LIN {X 0,Y 573.201,Z 603.99,A -85,B 0,C 180,E1 -2258.283,E2 -2258.283} C_VEL
LIN {X 0,Y 573.286,Z 595.539,A -85,B 0,C 180,E1 -2259.17,E2 -2259.17} C_VEL
LIN {X 0,Y 573.421,Z 585.099,A -85,B 0,C 180,E1 -2260.058,E2 -2260.058} C_VEL
LIN {X 0,Y 573.55,Z 573.353,A -85,B 0,C 180,E1 -2260.858,E2 -2260.858} C_VEL
LIN {X 0,Y 573.653,Z 562.283,A -85,B 0,C 180,E1 -2261.447,E2 -2261.447} C_VEL
LIN {X 0,Y 573.759,Z 549.174,A -85,B 0,C 180,E1 -2261.974,E2 -2261.974} C_VEL
LIN {X 0,Y 573.841,Z 536.522,A -85,B 0,C 180,E1 -2262.331,E2 -2262.331} C_VEL
LIN {X 0,Y 573.932,Z 523.316,A -85,B 0,C 180,E1 -2262.554,E2 -2262.554} C_VEL
LIN {X 0,Y 574.025,Z 427.51,A -85,B 0,C 180,E1 -2263.757,E2 -2263.757} C_VEL
LIN {X 0,Y 573.376,Z 423.284,A -85,B 0,C 180,E1 -2263.851,E2 -2263.851} C_VEL
LIN {X 0,Y 573.504,Z 405.17,A -85,B 0,C 180,E1 -2266.547,E2 -2266.547} C_VEL
LIN {X 0,Y 573.685,Z 388.232,A -85,B 0,C 180,E1 -2269.129,E2 -2269.129} C_VEL
LIN {X 0,Y 573.876,Z 371.34,A -85,B 0,C 180,E1 -2271.744,E2 -2271.744} C_VEL
LIN {X 0,Y 573.288,Z 367.673,A -85,B 0,C 180,E1 -2272.383,E2 -2272.383} C_VEL
LIN {X 0,Y 573.259,Z 367.581,A -85,B 0,C 180,E1 -2275.409,E2 -2275.409} C_VEL
LIN {X 0,Y 573.252,Z 367.576,A -85,B 0,C 180,E1 -2278.028,E2 -2278.028} C_VEL
LIN {X 0,Y 573.24,Z 367.576,A -85,B 0,C 180,E1 -2280.884,E2 -2280.884} C_VEL
LIN {X 0,Y 573.262,Z 367.58,A -85,B 0,C 180,E1 -2283.523,E2 -2283.523} C_VEL
LIN {X 0,Y 573.262,Z 367.573,A -85,B 0,C 180,E1 -2286.047,E2 -2286.047} C_VEL
LIN {X 0,Y 573.249,Z 367.575,A -85,B 0,C 180,E1 -2288.7,E2 -2288.7} C_VEL
LIN {X 0,Y 573.253,Z 367.577,A -85,B 0,C 180,E1 -2291.595,E2 -2291.595} C_VEL
LIN {X 0,Y 573.237,Z 367.575,A -85,B 0,C 180,E1 -2294.332,E2 -2294.332} C_VEL
LIN {X 0,Y 573.249,Z 367.58,A -85,B 0,C 180,E1 -2297.357,E2 -2297.357} C_VEL
LIN {X 0,Y 573.271,Z 367.575,A -85,B 0,C 180,E1 -2299.477,E2 -2299.477} C_VEL
LIN {X 0,Y 573.234,Z 367.575,A -85,B 0,C 180,E1 -2302.192,E2 -2302.192} C_VEL
LIN {X 0,Y 573.264,Z 367.578,A -85,B 0,C 180,E1 -2304.816,E2 -2304.816} C_VEL
LIN {X 0,Y 573.253,Z 367.577,A -85,B 0,C 180,E1 -2307.355,E2 -2307.355} C_VEL
LIN {X 0,Y 573.245,Z 367.574,A -85,B 0,C 180,E1 -2309.824,E2 -2309.824} C_VEL
LIN {X 0,Y 573.284,Z 367.571,A -85,B 0,C 180,E1 -2312.235,E2 -2312.235} C_VEL
LIN {X 0,Y 573.263,Z 367.577,A -85,B 0,C 180,E1 -2315.121,E2 -2315.121} C_VEL
LIN {X 0,Y 573.233,Z 367.576,A -85,B 0,C 180,E1 -2317.662,E2 -2317.662} C_VEL
LIN {X 0,Y 573.251,Z 367.574,A -85,B 0,C 180,E1 -2319.923,E2 -2319.923} C_VEL
LIN {X 0,Y 573.258,Z 367.578,A -85,B 0,C 180,E1 -2322.988,E2 -2322.988} C_VEL
LIN {X 0,Y 573.266,Z 367.572,A -85,B 0,C 180,E1 -2325.807,E2 -2325.807} C_VEL
LIN {X 0,Y 573.255,Z 367.58,A -85,B 0,C 180,E1 -2328.745,E2 -2328.745} C_VEL
LIN {X 0,Y 573.284,Z 367.569,A -85,B 0,C 180,E1 -2331.54,E2 -2331.54} C_VEL
LIN {X 0,Y 573.285,Z 367.578,A -85,B 0,C 180,E1 -2334.372,E2 -2334.372} C_VEL
LIN {X 0,Y 573.302,Z 367.57,A -85,B 0,C 180,E1 -2337.892,E2 -2337.892} C_VEL
LIN {X 0,Y 573.329,Z 367.568,A -85,B 0,C 180,E1 -2340.702,E2 -2340.702} C_VEL
LIN {X 0,Y 573.235,Z 367.576,A -85,B 0,C 180,E1 -2343.514,E2 -2343.514} C_VEL
LIN {X 0,Y 573.287,Z 367.57,A -85,B 0,C 180,E1 -2345.628,E2 -2345.628} C_VEL
LIN {X 0,Y 573.284,Z 367.576,A -85,B 0,C 180,E1 -2348.459,E2 -2348.459} C_VEL
LIN {X 0,Y 573.264,Z 367.572,A -85,B 0,C 180,E1 -2351.312,E2 -2351.312} C_VEL
LIN {X 0,Y 573.267,Z 367.58,A -85,B 0,C 180,E1 -2354.193,E2 -2354.193} C_VEL
LIN {X 0,Y 573.255,Z 367.573,A -85,B 0,C 180,E1 -2357.112,E2 -2357.112} C_VEL
LIN {X 0,Y 573.252,Z 367.582,A -85,B 0,C 180,E1 -2360.077,E2 -2360.077} C_VEL
LIN {X 0,Y 573.235,Z 367.58,A -85,B 0,C 180,E1 -2362.338,E2 -2362.338} C_VEL
LIN {X 0,Y 573.247,Z 367.576,A -85,B 0,C 180,E1 -2364.398,E2 -2364.398} C_VEL
LIN {X 0,Y 572.62,Z 367.654,A -85,B 0,C 180,E1 -2364.985,E2 -2364.985} C_VEL
LIN {X 0,Y 569.781,Z 368.014,A -85,B 0,C 180,E1 -2365.936,E2 -2365.936} C_VEL
LIN {X 0,Y 567.353,Z 368.314,A -85,B 0,C 180,E1 -2366.702,E2 -2366.702} C_VEL
LIN {X 0,Y 566.301,Z 368.442,A -85,B 0,C 180,E1 -2367.294,E2 -2367.294} C_VEL
LIN {X 0,Y 566.212,Z 368.452,A -85,B 0,C 180,E1 -2367.494,E2 -2367.494} C_VEL
LIN {X 0,Y 566.223,Z 368.458,A -85,B 0,C 180,E1 -2369.768,E2 -2369.768} C_VEL
LIN {X 0,Y 566.205,Z 368.453,A -85,B 0,C 180,E1 -2372.432,E2 -2372.432} C_VEL
LIN {X 0,Y 566.209,Z 368.452,A -85,B 0,C 180,E1 -2374.995,E2 -2374.995} C_VEL
LIN {X 0,Y 566.193,Z 368.459,A -85,B 0,C 180,E1 -2377.461,E2 -2377.461} C_VEL
LIN {X 0,Y 566.224,Z 368.451,A -85,B 0,C 180,E1 -2380.198,E2 -2380.198} C_VEL
LIN {X 0,Y 566.203,Z 368.454,A -85,B 0,C 180,E1 -2383.054,E2 -2383.054} C_VEL
LIN {X 0,Y 566.195,Z 368.455,A -85,B 0,C 180,E1 -2386.049,E2 -2386.049} C_VEL
LIN {X 0,Y 566.21,Z 368.452,A -85,B 0,C 180,E1 -2388.864,E2 -2388.864} C_VEL
LIN {X 0,Y 566.189,Z 368.46,A -85,B 0,C 180,E1 -2391.638,E2 -2391.638} C_VEL
LIN {X 0,Y 566.212,Z 368.45,A -85,B 0,C 180,E1 -2394.312,E2 -2394.312} C_VEL
LIN {X 0,Y 566.228,Z 368.451,A -85,B 0,C 180,E1 -2396.899,E2 -2396.899} C_VEL
LIN {X 0,Y 566.185,Z 368.461,A -85,B 0,C 180,E1 -2399.408,E2 -2399.408} C_VEL
LIN {X 0,Y 566.212,Z 368.452,A -85,B 0,C 180,E1 -2401.858,E2 -2401.858} C_VEL
LIN {X 0,Y 566.215,Z 368.45,A -85,B 0,C 180,E1 -2404.251,E2 -2404.251} C_VEL
LIN {X 0,Y 566.174,Z 368.458,A -85,B 0,C 180,E1 -2406.718,E2 -2406.718} C_VEL
LIN {X 0,Y 566.208,Z 368.452,A -85,B 0,C 180,E1 -2409.663,E2 -2409.663} C_VEL
LIN {X 0,Y 566.201,Z 368.455,A -85,B 0,C 180,E1 -2412.669,E2 -2412.669} C_VEL
LIN {X 0,Y 566.237,Z 368.449,A -85,B 0,C 180,E1 -2415.627,E2 -2415.627} C_VEL
LIN {X 0,Y 566.237,Z 368.453,A -85,B 0,C 180,E1 -2418.675,E2 -2418.675} C_VEL
LIN {X 0,Y 566.23,Z 368.454,A -85,B 0,C 180,E1 -2421.434,E2 -2421.434} C_VEL
LIN {X 0,Y 566.259,Z 368.58,A -85,B 0,C 180,E1 -2422.203,E2 -2422.203} C_VEL
LIN {X 0,Y 566.656,Z 372.244,A -85,B 0,C 180,E1 -2422.875,E2 -2422.875} C_VEL
LIN {X 0,Y 566.541,Z 387.974,A -85,B 0,C 180,E1 -2425.553,E2 -2425.553} C_VEL
LIN {X 0,Y 566.343,Z 407.089,A -85,B 0,C 180,E1 -2428.755,E2 -2428.755} C_VEL
LIN {X 0,Y 566.33,Z 408.914,A -85,B 0,C 180,E1 -2429.022,E2 -2429.022} C_VEL
LIN {X 0,Y 566.891,Z 412.581,A -85,B 0,C 180,E1 -2429.112,E2 -2429.112} C_VEL
LIN {X 0,Y 567.185,Z 418.987,A -85,B 0,C 180,E1 -2429.201,E2 -2429.201} C_VEL
LIN {X 0,Y 566.972,Z 515.705,A -85,B 0,C 180,E1 -2430.444,E2 -2430.444} C_VEL
LIN {X 0,Y 566.89,Z 528.87,A -85,B 0,C 180,E1 -2430.755,E2 -2430.755} C_VEL
LIN {X 0,Y 566.741,Z 541.512,A -85,B 0,C 180,E1 -2431.199,E2 -2431.199} C_VEL
LIN {X 0,Y 566.56,Z 553.601,A -85,B 0,C 180,E1 -2431.777,E2 -2431.777} C_VEL
LIN {X 0,Y 566.433,Z 565.04,A -85,B 0,C 180,E1 -2432.489,E2 -2432.489} C_VEL
LIN {X 0,Y 566.294,Z 575.37,A -85,B 0,C 180,E1 -2433.29,E2 -2433.29} C_VEL
LIN {X 0,Y 566.172,Z 583.857,A -85,B 0,C 180,E1 -2434.093,E2 -2434.093} C_VEL
LIN {X 0,Y 566.132,Z 591.698,A -85,B 0,C 180,E1 -2434.985,E2 -2434.985} C_VEL
LIN {X 0,Y 566.025,Z 599.41,A -85,B 0,C 180,E1 -2436.058,E2 -2436.058} C_VEL
LIN {X 0,Y 565.97,Z 605.612,A -85,B 0,C 180,E1 -2437.133,E2 -2437.133} C_VEL
LIN {X 0,Y 565.959,Z 610.553,A -85,B 0,C 180,E1 -2438.21,E2 -2438.21} C_VEL
LIN {X 0,Y 565.876,Z 614.383,A -85,B 0,C 180,E1 -2439.291,E2 -2439.291} C_VEL
LIN {X 0,Y 565.887,Z 616.355,A -85,B 0,C 180,E1 -2440.013,E2 -2440.013} C_VEL
LIN {X 0,Y 565.901,Z 618.581,A -85,B 0,C 180,E1 -2441.153,E2 -2441.153} C_VEL
LIN {X 0,Y 565.865,Z 619.69,A -85,B 0,C 180,E1 -2442.189,E2 -2442.189} C_VEL
LIN {X 0,Y 565.843,Z 619.978,A -85,B 0,C 180,E1 -2442.918,E2 -2442.918} C_VEL
LIN {X 0,Y 565.863,Z 619.855,A -85,B 0,C 180,E1 -2443.649,E2 -2443.649} C_VEL
LIN {X 0,Y 565.877,Z 619.281,A -85,B 0,C 180,E1 -2444.382,E2 -2444.382} C_VEL
LIN {X 0,Y 565.811,Z 618.293,A -85,B 0,C 180,E1 -2445.12,E2 -2445.12} C_VEL
LIN {X 0,Y 565.832,Z 616.886,A -85,B 0,C 180,E1 -2445.857,E2 -2445.857} C_VEL
LIN {X 0,Y 565.898,Z 613.759,A -85,B 0,C 180,E1 -2447.005,E2 -2447.005} C_VEL
LIN {X 0,Y 565.928,Z 609.725,A -85,B 0,C 180,E1 -2448.087,E2 -2448.087} C_VEL
LIN {X 0,Y 565.987,Z 603.691,A -85,B 0,C 180,E1 -2449.315,E2 -2449.315} C_VEL
LIN {X 0,Y 566.045,Z 596.024,A -85,B 0,C 180,E1 -2450.533,E2 -2450.533} C_VEL
LIN {X 0,Y 566.161,Z 587.806,A -85,B 0,C 180,E1 -2451.568,E2 -2451.568} C_VEL
LIN {X 0,Y 566.268,Z 578.376,A -85,B 0,C 180,E1 -2452.531,E2 -2452.531} C_VEL
LIN {X 0,Y 566.386,Z 567.954,A -85,B 0,C 180,E1 -2453.395,E2 -2453.395} C_VEL
LIN {X 0,Y 566.546,Z 556.203,A -85,B 0,C 180,E1 -2454.164,E2 -2454.164} C_VEL
LIN {X 0,Y 566.673,Z 543.843,A -85,B 0,C 180,E1 -2454.793,E2 -2454.793} C_VEL
LIN {X 0,Y 566.851,Z 531.171,A -85,B 0,C 180,E1 -2455.268,E2 -2455.268} C_VEL
LIN {X 0,Y 566.956,Z 517.562,A -85,B 0,C 180,E1 -2455.61,E2 -2455.61} C_VEL
LIN {X 0,Y 567.038,Z 490.594,A -85,B 0,C 180,E1 -2455.979,E2 -2455.979} C_VEL
LIN {X 0,Y 567.083,Z 413.826,A -85,B 0,C 180,E1 -2456.957,E2 -2456.957} C_VEL
LIN {X 0,Y 566.313,Z 409.219,A -85,B 0,C 180,E1 -2457.05,E2 -2457.05} C_VEL
LIN {X 0,Y 566.268,Z 407.096,A -85,B 0,C 180,E1 -2457.335,E2 -2457.335} C_VEL
LIN {X 0,Y 566.476,Z 390.202,A -85,B 0,C 180,E1 -2460.162,E2 -2460.162} C_VEL
LIN {X 0,Y 566.678,Z 373.075,A -85,B 0,C 180,E1 -2463.071,E2 -2463.071} C_VEL
LIN {X 0,Y 566.23,Z 368.551,A -85,B 0,C 180,E1 -2463.903,E2 -2463.903} C_VEL
LIN {X 0,Y 566.214,Z 368.453,A -85,B 0,C 180,E1 -2466.568,E2 -2466.568} C_VEL
LIN {X 0,Y 566.21,Z 368.453,A -85,B 0,C 180,E1 -2469.685,E2 -2469.685} C_VEL
LIN {X 0,Y 566.21,Z 368.451,A -85,B 0,C 180,E1 -2472.086,E2 -2472.086} C_VEL
LIN {X 0,Y 566.169,Z 368.464,A -85,B 0,C 180,E1 -2475.035,E2 -2475.035} C_VEL
LIN {X 0,Y 566.225,Z 368.447,A -85,B 0,C 180,E1 -2478.134,E2 -2478.134} C_VEL
LIN {X 0,Y 566.218,Z 368.453,A -85,B 0,C 180,E1 -2480.727,E2 -2480.727} C_VEL
LIN {X 0,Y 566.212,Z 368.45,A -85,B 0,C 180,E1 -2483.783,E2 -2483.783} C_VEL
LIN {X 0,Y 566.222,Z 368.448,A -85,B 0,C 180,E1 -2486.262,E2 -2486.262} C_VEL
LIN {X 0,Y 566.197,Z 368.46,A -85,B 0,C 180,E1 -2488.92,E2 -2488.92} C_VEL
LIN {X 0,Y 566.192,Z 368.46,A -85,B 0,C 180,E1 -2491.047,E2 -2491.047} C_VEL
LIN {X 0,Y 566.24,Z 368.449,A -85,B 0,C 180,E1 -2493.46,E2 -2493.46} C_VEL
LIN {X 0,Y 566.197,Z 368.452,A -85,B 0,C 180,E1 -2495.819,E2 -2495.819} C_VEL
LIN {X 0,Y 566.209,Z 368.458,A -85,B 0,C 180,E1 -2498.902,E2 -2498.902} C_VEL
LIN {X 0,Y 566.206,Z 368.456,A -85,B 0,C 180,E1 -2501.172,E2 -2501.172} C_VEL
LIN {X 0,Y 566.215,Z 368.452,A -85,B 0,C 180,E1 -2503.412,E2 -2503.412} C_VEL
LIN {X 0,Y 566.195,Z 368.453,A -85,B 0,C 180,E1 -2506.359,E2 -2506.359} C_VEL
LIN {X 0,Y 566.265,Z 368.449,A -85,B 0,C 180,E1 -2508.654,E2 -2508.654} C_VEL
LIN {X 0,Y 566.242,Z 368.448,A -85,B 0,C 180,E1 -2511.435,E2 -2511.435} C_VEL
LIN {X 0,Y 566.256,Z 368.445,A -85,B 0,C 180,E1 -2514.302,E2 -2514.302} C_VEL
LIN {X 0,Y 566.272,Z 368.442,A -85,B 0,C 180,E1 -2517.866,E2 -2517.866} C_VEL
LIN {X 0,Y 566.303,Z 368.446,A -85,B 0,C 180,E1 -2520.711,E2 -2520.711} C_VEL
LIN {X 0,Y 566.274,Z 368.45,A -85,B 0,C 180,E1 -2522.846,E2 -2522.846} C_VEL
LIN {X 0,Y 566.254,Z 368.444,A -85,B 0,C 180,E1 -2525.698,E2 -2525.698} C_VEL
LIN {X 0,Y 566.241,Z 368.452,A -85,B 0,C 180,E1 -2528.566,E2 -2528.566} C_VEL
LIN {X 0,Y 566.242,Z 368.447,A -85,B 0,C 180,E1 -2531.454,E2 -2531.454} C_VEL
LIN {X 0,Y 566.224,Z 368.453,A -85,B 0,C 180,E1 -2534.507,E2 -2534.507} C_VEL
LIN {X 0,Y 566.197,Z 368.452,A -85,B 0,C 180,E1 -2537.332,E2 -2537.332} C_VEL
LIN {X 0,Y 566.213,Z 368.453,A -85,B 0,C 180,E1 -2540.337,E2 -2540.337} C_VEL
LIN {X 0,Y 566.222,Z 368.449,A -85,B 0,C 180,E1 -2543.403,E2 -2543.403} C_VEL
LIN {X 0,Y 566.218,Z 368.449,A -85,B 0,C 180,E1 -2545.749,E2 -2545.749} C_VEL
LIN {X 0,Y 566.201,Z 368.454,A -85,B 0,C 180,E1 -2548.204,E2 -2548.204} C_VEL
LIN {X 0,Y 566.193,Z 368.455,A -85,B 0,C 180,E1 -2551.079,E2 -2551.079} C_VEL
LIN {X 0,Y 566.223,Z 368.448,A -85,B 0,C 180,E1 -2553.738,E2 -2553.738} C_VEL
LIN {X 0,Y 566.211,Z 368.46,A -85,B 0,C 180,E1 -2556.569,E2 -2556.569} C_VEL
LIN {X 0,Y 566.209,Z 368.45,A -85,B 0,C 180,E1 -2559.687,E2 -2559.687} C_VEL
LIN {X 0,Y 566.216,Z 368.449,A -85,B 0,C 180,E1 -2562.087,E2 -2562.087} C_VEL
LIN {X 0,Y 566.169,Z 368.457,A -85,B 0,C 180,E1 -2565.037,E2 -2565.037} C_VEL
LIN {X 0,Y 566.215,Z 368.453,A -85,B 0,C 180,E1 -2568.137,E2 -2568.137} C_VEL
LIN {X 0,Y 566.22,Z 368.455,A -85,B 0,C 180,E1 -2570.728,E2 -2570.728} C_VEL
LIN {X 0,Y 566.217,Z 368.449,A -85,B 0,C 180,E1 -2573.784,E2 -2573.784} C_VEL
LIN {X 0,Y 566.229,Z 368.454,A -85,B 0,C 180,E1 -2576.264,E2 -2576.264} C_VEL
LIN {X 0,Y 566.199,Z 368.455,A -85,B 0,C 180,E1 -2578.923,E2 -2578.923} C_VEL
LIN {X 0,Y 566.229,Z 368.45,A -85,B 0,C 180,E1 -2581.859,E2 -2581.859} C_VEL
LIN {X 0,Y 566.226,Z 368.457,A -85,B 0,C 180,E1 -2584.252,E2 -2584.252} C_VEL
LIN {X 0,Y 566.243,Z 368.528,A -85,B 0,C 180,E1 -2587.468,E2 -2587.468} C_VEL
LIN {X 0,Y 566.914,Z 372.503,A -85,B 0,C 180,E1 -2588.167,E2 -2588.167} C_VEL
LIN {X 0,Y 566.728,Z 389.583,A -85,B 0,C 180,E1 -2590.837,E2 -2590.837} C_VEL
LIN {X 0,Y 566.496,Z 406.333,A -85,B 0,C 180,E1 -2593.421,E2 -2593.421} C_VEL
LIN {X 0,Y 566.375,Z 423.296,A -85,B 0,C 180,E1 -2595.975,E2 -2595.975} C_VEL
LIN {X 0,Y 567.201,Z 430.334,A -85,B 0,C 180,E1 -2596.11,E2 -2596.11} C_VEL
LIN {X 0,Y 566.982,Z 530.968,A -85,B 0,C 180,E1 -2597.404,E2 -2597.404} C_VEL
LIN {X 0,Y 566.887,Z 544.233,A -85,B 0,C 180,E1 -2597.72,E2 -2597.72} C_VEL
LIN {X 0,Y 566.745,Z 556.386,A -85,B 0,C 180,E1 -2598.149,E2 -2598.149} C_VEL
LIN {X 0,Y 566.627,Z 568.16,A -85,B 0,C 180,E1 -2598.709,E2 -2598.709} C_VEL
LIN {X 0,Y 566.485,Z 578.914,A -85,B 0,C 180,E1 -2599.366,E2 -2599.366} C_VEL
LIN {X 0,Y 566.332,Z 589.545,A -85,B 0,C 180,E1 -2600.176,E2 -2600.176} C_VEL
LIN {X 0,Y 566.207,Z 599.116,A -85,B 0,C 180,E1 -2601.075,E2 -2601.075} C_VEL
LIN {X 0,Y 566.112,Z 606.963,A -85,B 0,C 180,E1 -2601.972,E2 -2601.972} C_VEL
LIN {X 0,Y 566.003,Z 614.624,A -85,B 0,C 180,E1 -2603.047,E2 -2603.047} C_VEL
LIN {X 0,Y 566.004,Z 621.681,A -85,B 0,C 180,E1 -2604.299,E2 -2604.299} C_VEL
LIN {X 0,Y 565.933,Z 626.373,A -85,B 0,C 180,E1 -2605.37,E2 -2605.37} C_VEL
LIN {X 0,Y 565.927,Z 629.958,A -85,B 0,C 180,E1 -2606.44,E2 -2606.44} C_VEL
LIN {X 0,Y 565.878,Z 631.808,A -85,B 0,C 180,E1 -2607.153,E2 -2607.153} C_VEL
LIN {X 0,Y 565.846,Z 634.185,A -85,B 0,C 180,E1 -2608.577,E2 -2608.577} C_VEL
LIN {X 0,Y 565.839,Z 635,A -85,B 0,C 180,E1 -2610,E2 -2610} C_VEL
LIN {X 0,Y 565.846,Z 634.186,A -85,B 0,C 180,E1 -2611.424,E2 -2611.424} C_VEL
LIN {X 0,Y 565.878,Z 631.81,A -85,B 0,C 180,E1 -2612.848,E2 -2612.848} C_VEL
LIN {X 0,Y 565.926,Z 628.895,A -85,B 0,C 180,E1 -2613.917,E2 -2613.917} C_VEL
LIN {X 0,Y 565.878,Z 624.948,A -85,B 0,C 180,E1 -2614.988,E2 -2614.988} C_VEL
LIN {X 0,Y 566.002,Z 619.867,A -85,B 0,C 180,E1 -2616.059,E2 -2616.059} C_VEL
LIN {X 0,Y 566.04,Z 613.468,A -85,B 0,C 180,E1 -2617.132,E2 -2617.132} C_VEL
LIN {X 0,Y 566.134,Z 605.478,A -85,B 0,C 180,E1 -2618.208,E2 -2618.208} C_VEL
LIN {X 0,Y 566.228,Z 597.335,A -85,B 0,C 180,E1 -2619.105,E2 -2619.105} C_VEL
LIN {X 0,Y 566.342,Z 587.4,A -85,B 0,C 180,E1 -2620.005,E2 -2620.005} C_VEL
LIN {X 0,Y 566.525,Z 576.286,A -85,B 0,C 180,E1 -2620.808,E2 -2620.808} C_VEL
LIN {X 0,Y 566.66,Z 565.177,A -85,B 0,C 180,E1 -2621.446,E2 -2621.446} C_VEL
LIN {X 0,Y 566.748,Z 552.984,A -85,B 0,C 180,E1 -2621.988,E2 -2621.988} C_VEL
LIN {X 0,Y 566.892,Z 540.179,A -85,B 0,C 180,E1 -2622.394,E2 -2622.394} C_VEL
LIN {X 0,Y 566.999,Z 526.607,A -85,B 0,C 180,E1 -2622.664,E2 -2622.664} C_VEL
LIN {X 0,Y 567.041,Z 427.835,A -85,B 0,C 180,E1 -2623.926,E2 -2623.926} C_VEL
LIN {X 0,Y 566.373,Z 423.294,A -85,B 0,C 180,E1 -2624.026,E2 -2624.026} C_VEL
LIN {X 0,Y 566.532,Z 404.242,A -85,B 0,C 180,E1 -2626.899,E2 -2626.899} C_VEL
LIN {X 0,Y 566.748,Z 387.025,A -85,B 0,C 180,E1 -2629.561,E2 -2629.561} C_VEL
LIN {X 0,Y 566.915,Z 372.504,A -85,B 0,C 180,E1 -2631.833,E2 -2631.833} C_VEL
LIN {X 0,Y 566.244,Z 368.526,A -85,B 0,C 180,E1 -2632.532,E2 -2632.532} C_VEL
LIN {X 0,Y 566.218,Z 368.456,A -85,B 0,C 180,E1 -2635.748,E2 -2635.748} C_VEL
LIN {X 0,Y 566.204,Z 368.452,A -85,B 0,C 180,E1 -2638.202,E2 -2638.202} C_VEL
LIN {X 0,Y 566.201,Z 368.455,A -85,B 0,C 180,E1 -2641.077,E2 -2641.077} C_VEL
LIN {X 0,Y 566.213,Z 368.454,A -85,B 0,C 180,E1 -2643.734,E2 -2643.734} C_VEL
LIN {X 0,Y 566.217,Z 368.45,A -85,B 0,C 180,E1 -2646.568,E2 -2646.568} C_VEL
LIN {X 0,Y 566.213,Z 368.454,A -85,B 0,C 180,E1 -2649.685,E2 -2649.685} C_VEL
LIN {X 0,Y 566.213,Z 368.45,A -85,B 0,C 180,E1 -2652.087,E2 -2652.087} C_VEL
LIN {X 0,Y 566.172,Z 368.462,A -85,B 0,C 180,E1 -2655.035,E2 -2655.035} C_VEL
LIN {X 0,Y 566.224,Z 368.449,A -85,B 0,C 180,E1 -2658.134,E2 -2658.134} C_VEL
LIN {X 0,Y 566.221,Z 368.453,A -85,B 0,C 180,E1 -2660.727,E2 -2660.727} C_VEL
LIN {X 0,Y 566.215,Z 368.451,A -85,B 0,C 180,E1 -2663.783,E2 -2663.783} C_VEL
LIN {X 0,Y 566.208,Z 368.452,A -85,B 0,C 180,E1 -2666.265,E2 -2666.265} C_VEL
LIN {X 0,Y 566.195,Z 368.461,A -85,B 0,C 180,E1 -2668.921,E2 -2668.921} C_VEL
LIN {X 0,Y 566.223,Z 368.449,A -85,B 0,C 180,E1 -2671.858,E2 -2671.858} C_VEL
LIN {X 0,Y 566.219,Z 368.451,A -85,B 0,C 180,E1 -2674.251,E2 -2674.251} C_VEL
LIN {X 0,Y 566.185,Z 368.461,A -85,B 0,C 180,E1 -2676.713,E2 -2676.713} C_VEL
LIN {X 0,Y 566.214,Z 368.45,A -85,B 0,C 180,E1 -2679.663,E2 -2679.663} C_VEL
LIN {X 0,Y 566.199,Z 368.46,A -85,B 0,C 180,E1 -2682.668,E2 -2682.668} C_VEL
LIN {X 0,Y 566.227,Z 368.449,A -85,B 0,C 180,E1 -2685.627,E2 -2685.627} C_VEL
LIN {X 0,Y 566.227,Z 368.457,A -85,B 0,C 180,E1 -2688.675,E2 -2688.675} C_VEL
LIN {X 0,Y 566.228,Z 368.449,A -85,B 0,C 180,E1 -2691.434,E2 -2691.434} C_VEL
LIN {X 0,Y 566.253,Z 368.452,A -85,B 0,C 180,E1 -2694.302,E2 -2694.302} C_VEL
LIN {X 0,Y 566.273,Z 368.445,A -85,B 0,C 180,E1 -2697.866,E2 -2697.866} C_VEL
LIN {X 0,Y 566.299,Z 368.444,A -85,B 0,C 180,E1 -2700.711,E2 -2700.711} C_VEL
LIN {X 0,Y 566.271,Z 368.446,A -85,B 0,C 180,E1 -2702.846,E2 -2702.846} C_VEL
LIN {X 0,Y 566.255,Z 368.447,A -85,B 0,C 180,E1 -2705.698,E2 -2705.698} C_VEL
LIN {X 0,Y 566.228,Z 368.453,A -85,B 0,C 180,E1 -2708.566,E2 -2708.566} C_VEL
LIN {X 0,Y 566.235,Z 368.449,A -85,B 0,C 180,E1 -2711.454,E2 -2711.454} C_VEL
LIN {X 0,Y 566.227,Z 368.453,A -85,B 0,C 180,E1 -2714.507,E2 -2714.507} C_VEL
LIN {X 0,Y 566.199,Z 368.453,A -85,B 0,C 180,E1 -2717.332,E2 -2717.332} C_VEL
LIN {X 0,Y 566.214,Z 368.455,A -85,B 0,C 180,E1 -2720.337,E2 -2720.337} C_VEL
LIN {X 0,Y 566.185,Z 368.456,A -85,B 0,C 180,E1 -2723.404,E2 -2723.404} C_VEL
LIN {X 0,Y 566.221,Z 368.457,A -85,B 0,C 180,E1 -2725.749,E2 -2725.749} C_VEL
LIN {X 0,Y 566.212,Z 368.452,A -85,B 0,C 180,E1 -2727.494,E2 -2727.494} C_VEL
LIN {X 0,Y 565.534,Z 368.542,A -85,B 0,C 180,E1 -2728.088,E2 -2728.088} C_VEL
LIN {X 0,Y 562.669,Z 368.895,A -85,B 0,C 180,E1 -2729.051,E2 -2729.051} C_VEL
LIN {X 0,Y 560.258,Z 369.2,A -85,B 0,C 180,E1 -2729.827,E2 -2729.827} C_VEL
LIN {X 0,Y 559.229,Z 369.323,A -85,B 0,C 180,E1 -2730.426,E2 -2730.426} C_VEL
LIN {X 0,Y 559.148,Z 369.331,A -85,B 0,C 180,E1 -2730.628,E2 -2730.628} C_VEL
LIN {X 0,Y 559.174,Z 369.334,A -85,B 0,C 180,E1 -2733.574,E2 -2733.574} C_VEL
LIN {X 0,Y 559.165,Z 369.329,A -85,B 0,C 180,E1 -2736.449,E2 -2736.449} C_VEL
LIN {X 0,Y 559.175,Z 369.328,A -85,B 0,C 180,E1 -2738.934,E2 -2738.934} C_VEL
LIN {X 0,Y 559.189,Z 369.332,A -85,B 0,C 180,E1 -2741.768,E2 -2741.768} C_VEL
LIN {X 0,Y 559.137,Z 369.332,A -85,B 0,C 180,E1 -2744.74,E2 -2744.74} C_VEL
LIN {X 0,Y 559.174,Z 369.332,A -85,B 0,C 180,E1 -2747.863,E2 -2747.863} C_VEL
LIN {X 0,Y 559.185,Z 369.327,A -85,B 0,C 180,E1 -2750.136,E2 -2750.136} C_VEL
LIN {X 0,Y 559.146,Z 369.333,A -85,B 0,C 180,E1 -2752.893,E2 -2752.893} C_VEL
LIN {X 0,Y 559.157,Z 369.336,A -85,B 0,C 180,E1 -2755.557,E2 -2755.557} C_VEL
LIN {X 0,Y 559.168,Z 369.328,A -85,B 0,C 180,E1 -2758.138,E2 -2758.138} C_VEL
LIN {X 0,Y 559.144,Z 369.332,A -85,B 0,C 180,E1 -2760.647,E2 -2760.647} C_VEL
LIN {X 0,Y 559.171,Z 369.336,A -85,B 0,C 180,E1 -2763.173,E2 -2763.173} C_VEL
LIN {X 0,Y 559.158,Z 369.334,A -85,B 0,C 180,E1 -2765.495,E2 -2765.495} C_VEL
LIN {X 0,Y 559.173,Z 369.329,A -85,B 0,C 180,E1 -2768.624,E2 -2768.624} C_VEL
LIN {X 0,Y 559.164,Z 369.335,A -85,B 0,C 180,E1 -2770.926,E2 -2770.926} C_VEL
LIN {X 0,Y 559.166,Z 369.328,A -85,B 0,C 180,E1 -2773.948,E2 -2773.948} C_VEL
LIN {X 0,Y 559.174,Z 369.327,A -85,B 0,C 180,E1 -2776.184,E2 -2776.184} C_VEL
LIN {X 0,Y 559.197,Z 369.332,A -85,B 0,C 180,E1 -2779.134,E2 -2779.134} C_VEL
LIN {X 0,Y 559.213,Z 369.481,A -85,B 0,C 180,E1 -2782.079,E2 -2782.079} C_VEL
LIN {X 0,Y 559.69,Z 373.303,A -85,B 0,C 180,E1 -2782.786,E2 -2782.786} C_VEL
LIN {X 0,Y 559.582,Z 384.755,A -85,B 0,C 180,E1 -2784.776,E2 -2784.776} C_VEL
LIN {X 0,Y 559.354,Z 401.688,A -85,B 0,C 180,E1 -2787.66,E2 -2787.66} C_VEL
LIN {X 0,Y 559.316,Z 408.773,A -85,B 0,C 180,E1 -2788.83,E2 -2788.83} C_VEL
LIN {X 0,Y 559.656,Z 411.132,A -85,B 0,C 180,E1 -2788.909,E2 -2788.909} C_VEL
LIN {X 0,Y 560.299,Z 416.022,A -85,B 0,C 180,E1 -2788.989,E2 -2788.989} C_VEL
LIN {X 0,Y 560.059,Z 516.026,A -85,B 0,C 180,E1 -2790.292,E2 -2790.292} C_VEL
LIN {X 0,Y 559.95,Z 529.093,A -85,B 0,C 180,E1 -2790.607,E2 -2790.607} C_VEL
LIN {X 0,Y 559.77,Z 542.238,A -85,B 0,C 180,E1 -2791.079,E2 -2791.079} C_VEL
LIN {X 0,Y 559.595,Z 553.326,A -85,B 0,C 180,E1 -2791.619,E2 -2791.619} C_VEL
LIN {X 0,Y 559.458,Z 564.814,A -85,B 0,C 180,E1 -2792.34,E2 -2792.34} C_VEL
LIN {X 0,Y 559.259,Z 575.199,A -85,B 0,C 180,E1 -2793.151,E2 -2793.151} C_VEL
LIN {X 0,Y 559.127,Z 583.711,A -85,B 0,C 180,E1 -2793.964,E2 -2793.964} C_VEL
LIN {X 0,Y 559.059,Z 591.577,A -85,B 0,C 180,E1 -2794.867,E2 -2794.867} C_VEL
LIN {X 0,Y 558.977,Z 599.313,A -85,B 0,C 180,E1 -2795.954,E2 -2795.954} C_VEL
LIN {X 0,Y 558.891,Z 606.441,A -85,B 0,C 180,E1 -2797.224,E2 -2797.224} C_VEL
LIN {X 0,Y 558.847,Z 611.21,A -85,B 0,C 180,E1 -2798.315,E2 -2798.315} C_VEL
LIN {X 0,Y 558.778,Z 614.874,A -85,B 0,C 180,E1 -2799.41,E2 -2799.41} C_VEL
LIN {X 0,Y 558.783,Z 616.764,A -85,B 0,C 180,E1 -2800.141,E2 -2800.141} C_VEL
LIN {X 0,Y 558.798,Z 618.666,A -85,B 0,C 180,E1 -2801.185,E2 -2801.185} C_VEL
LIN {X 0,Y 558.771,Z 619.8,A -85,B 0,C 180,E1 -2802.346,E2 -2802.346} C_VEL
LIN {X 0,Y 558.743,Z 619.997,A -85,B 0,C 180,E1 -2803.085,E2 -2803.085} C_VEL
LIN {X 0,Y 558.79,Z 619.245,A -85,B 0,C 180,E1 -2804.432,E2 -2804.432} C_VEL
LIN {X 0,Y 558.718,Z 618.026,A -85,B 0,C 180,E1 -2805.316,E2 -2805.316} C_VEL
LIN {X 0,Y 558.789,Z 615.557,A -85,B 0,C 180,E1 -2806.438,E2 -2806.438} C_VEL
LIN {X 0,Y 558.816,Z 612.008,A -85,B 0,C 180,E1 -2807.567,E2 -2807.567} C_VEL
LIN {X 0,Y 558.889,Z 607.258,A -85,B 0,C 180,E1 -2808.702,E2 -2808.702} C_VEL
LIN {X 0,Y 558.943,Z 601.108,A -85,B 0,C 180,E1 -2809.845,E2 -2809.845} C_VEL
LIN {X 0,Y 559.019,Z 593.325,A -85,B 0,C 180,E1 -2810.995,E2 -2810.995} C_VEL
LIN {X 0,Y 559.135,Z 585.12,A -85,B 0,C 180,E1 -2811.977,E2 -2811.977} C_VEL
LIN {X 0,Y 559.293,Z 575.347,A -85,B 0,C 180,E1 -2812.925,E2 -2812.925} C_VEL
LIN {X 0,Y 559.457,Z 564.111,A -85,B 0,C 180,E1 -2813.8,E2 -2813.8} C_VEL
LIN {X 0,Y 559.635,Z 553.112,A -85,B 0,C 180,E1 -2814.482,E2 -2814.482} C_VEL
LIN {X 0,Y 559.799,Z 540.824,A -85,B 0,C 180,E1 -2815.069,E2 -2815.069} C_VEL
LIN {X 0,Y 559.981,Z 527.634,A -85,B 0,C 180,E1 -2815.527,E2 -2815.527} C_VEL
LIN {X 0,Y 560.035,Z 514.835,A -85,B 0,C 180,E1 -2815.82,E2 -2815.82} C_VEL
LIN {X 0,Y 560.209,Z 414.702,A -85,B 0,C 180,E1 -2817.12,E2 -2817.12} C_VEL
LIN {X 0,Y 559.268,Z 409.016,A -85,B 0,C 180,E1 -2817.242,E2 -2817.242} C_VEL
LIN {X 0,Y 559.299,Z 404.78,A -85,B 0,C 180,E1 -2817.908,E2 -2817.908} C_VEL
LIN {X 0,Y 559.503,Z 387.838,A -85,B 0,C 180,E1 -2820.787,E2 -2820.787} C_VEL
LIN {X 0,Y 559.75,Z 373.215,A -85,B 0,C 180,E1 -2823.318,E2 -2823.318} C_VEL
LIN {X 0,Y 559.187,Z 369.388,A -85,B 0,C 180,E1 -2824.061,E2 -2824.061} C_VEL
LIN {X 0,Y 559.145,Z 369.339,A -85,B 0,C 180,E1 -2827.107,E2 -2827.107} C_VEL
LIN {X 0,Y 559.167,Z 369.329,A -85,B 0,C 180,E1 -2829.942,E2 -2829.942} C_VEL
LIN {X 0,Y 559.159,Z 369.333,A -85,B 0,C 180,E1 -2832.742,E2 -2832.742} C_VEL
LIN {X 0,Y 559.15,Z 369.331,A -85,B 0,C 180,E1 -2835.76,E2 -2835.76} C_VEL
LIN {X 0,Y 559.197,Z 369.322,A -85,B 0,C 180,E1 -2838.233,E2 -2838.233} C_VEL
LIN {X 0,Y 559.173,Z 369.334,A -85,B 0,C 180,E1 -2841.19,E2 -2841.19} C_VEL
LIN {X 0,Y 559.166,Z 369.328,A -85,B 0,C 180,E1 -2843.791,E2 -2843.791} C_VEL
LIN {X 0,Y 559.171,Z 369.327,A -85,B 0,C 180,E1 -2846.426,E2 -2846.426} C_VEL
LIN {X 0,Y 559.161,Z 369.336,A -85,B 0,C 180,E1 -2848.981,E2 -2848.981} C_VEL
LIN {X 0,Y 559.164,Z 369.329,A -85,B 0,C 180,E1 -2851.617,E2 -2851.617} C_VEL
LIN {X 0,Y 559.193,Z 369.324,A -85,B 0,C 180,E1 -2853.904,E2 -2853.904} C_VEL
LIN {X 0,Y 559.155,Z 369.336,A -85,B 0,C 180,E1 -2857.068,E2 -2857.068} C_VEL
LIN {X 0,Y 559.179,Z 369.329,A -85,B 0,C 180,E1 -2859.395,E2 -2859.395} C_VEL
LIN {X 0,Y 559.148,Z 369.329,A -85,B 0,C 180,E1 -2861.686,E2 -2861.686} C_VEL
LIN {X 0,Y 559.165,Z 369.327,A -85,B 0,C 180,E1 -2863.948,E2 -2863.948} C_VEL
LIN {X 0,Y 559.167,Z 369.327,A -85,B 0,C 180,E1 -2866.184,E2 -2866.184} C_VEL
LIN {X 0,Y 559.203,Z 369.327,A -85,B 0,C 180,E1 -2869.134,E2 -2869.134} C_VEL
LIN {X 0,Y 559.205,Z 369.323,A -85,B 0,C 180,E1 -2872.054,E2 -2872.054} C_VEL
LIN {X 0,Y 559.252,Z 369.325,A -85,B 0,C 180,E1 -2874.953,E2 -2874.953} C_VEL
LIN {X 0,Y 559.244,Z 369.317,A -85,B 0,C 180,E1 -2877.839,E2 -2877.839} C_VEL
LIN {X 0,Y 559.272,Z 369.321,A -85,B 0,C 180,E1 -2880.72,E2 -2880.72} C_VEL
LIN {X 0,Y 559.239,Z 369.325,A -85,B 0,C 180,E1 -2882.881,E2 -2882.881} C_VEL
LIN {X 0,Y 559.223,Z 369.32,A -85,B 0,C 180,E1 -2885.77,E2 -2885.77} C_VEL
LIN {X 0,Y 559.196,Z 369.331,A -85,B 0,C 180,E1 -2888.674,E2 -2888.674} C_VEL
LIN {X 0,Y 559.2,Z 369.323,A -85,B 0,C 180,E1 -2891.601,E2 -2891.601} C_VEL
LIN {X 0,Y 559.189,Z 369.33,A -85,B 0,C 180,E1 -2894.596,E2 -2894.596} C_VEL
LIN {X 0,Y 559.157,Z 369.328,A -85,B 0,C 180,E1 -2897.557,E2 -2897.557} C_VEL
LIN {X 0,Y 559.167,Z 369.327,A -85,B 0,C 180,E1 -2899.838,E2 -2899.838} C_VEL
LIN {X 0,Y 559.148,Z 369.331,A -85,B 0,C 180,E1 -2902.153,E2 -2902.153} C_VEL
LIN {X 0,Y 559.153,Z 369.336,A -85,B 0,C 180,E1 -2904.505,E2 -2904.505} C_VEL
LIN {X 0,Y 559.173,Z 369.332,A -85,B 0,C 180,E1 -2906.902,E2 -2906.902} C_VEL
LIN {X 0,Y 559.143,Z 369.33,A -85,B 0,C 180,E1 -2909.859,E2 -2909.859} C_VEL
LIN {X 0,Y 559.17,Z 369.335,A -85,B 0,C 180,E1 -2912.715,E2 -2912.715} C_VEL
LIN {X 0,Y 559.152,Z 369.33,A -85,B 0,C 180,E1 -2915.322,E2 -2915.322} C_VEL
LIN {X 0,Y 559.13,Z 369.333,A -85,B 0,C 180,E1 -2918.018,E2 -2918.018} C_VEL
LIN {X 0,Y 559.175,Z 369.328,A -85,B 0,C 180,E1 -2920.811,E2 -2920.811} C_VEL
LIN {X 0,Y 559.16,Z 369.329,A -85,B 0,C 180,E1 -2923.732,E2 -2923.732} C_VEL
LIN {X 0,Y 559.164,Z 369.333,A -85,B 0,C 180,E1 -2926.802,E2 -2926.802} C_VEL
LIN {X 0,Y 559.174,Z 369.327,A -85,B 0,C 180,E1 -2929.19,E2 -2929.19} C_VEL
LIN {X 0,Y 559.133,Z 369.334,A -85,B 0,C 180,E1 -2931.984,E2 -2931.984} C_VEL
LIN {X 0,Y 559.16,Z 369.333,A -85,B 0,C 180,E1 -2934.784,E2 -2934.784} C_VEL
LIN {X 0,Y 559.173,Z 369.327,A -85,B 0,C 180,E1 -2937.362,E2 -2937.362} C_VEL
LIN {X 0,Y 559.15,Z 369.336,A -85,B 0,C 180,E1 -2940.143,E2 -2940.143} C_VEL
LIN {X 0,Y 559.182,Z 369.328,A -85,B 0,C 180,E1 -2943.171,E2 -2943.171} C_VEL
LIN {X 0,Y 559.158,Z 369.332,A -85,B 0,C 180,E1 -2945.496,E2 -2945.496} C_VEL
LIN {X 0,Y 559.187,Z 369.502,A -85,B 0,C 180,E1 -2947.363,E2 -2947.363} C_VEL
LIN {X 0,Y 559.973,Z 375.381,A -85,B 0,C 180,E1 -2948.355,E2 -2948.355} C_VEL
LIN {X 0,Y 559.721,Z 393.057,A -85,B 0,C 180,E1 -2951.137,E2 -2951.137} C_VEL
LIN {X 0,Y 559.478,Z 409.953,A -85,B 0,C 180,E1 -2953.77,E2 -2953.77} C_VEL
LIN {X 0,Y 559.387,Z 423.305,A -85,B 0,C 180,E1 -2955.796,E2 -2955.796} C_VEL
LIN {X 0,Y 560.301,Z 430.334,A -85,B 0,C 180,E1 -2955.935,E2 -2955.935} C_VEL
LIN {X 0,Y 560.075,Z 530.968,A -85,B 0,C 180,E1 -2957.246,E2 -2957.246} C_VEL
LIN {X 0,Y 559.935,Z 544.232,A -85,B 0,C 180,E1 -2957.565,E2 -2957.565} C_VEL
LIN {X 0,Y 559.793,Z 556.388,A -85,B 0,C 180,E1 -2957.999,E2 -2957.999} C_VEL
LIN {X 0,Y 559.668,Z 567.818,A -85,B 0,C 180,E1 -2958.548,E2 -2958.548} C_VEL
LIN {X 0,Y 559.499,Z 578.912,A -85,B 0,C 180,E1 -2959.231,E2 -2959.231} C_VEL
LIN {X 0,Y 559.313,Z 589.543,A -85,B 0,C 180,E1 -2960.051,E2 -2960.051} C_VEL
LIN {X 0,Y 559.161,Z 599.116,A -85,B 0,C 180,E1 -2960.961,E2 -2960.961} C_VEL
LIN {X 0,Y 559.05,Z 606.963,A -85,B 0,C 180,E1 -2961.87,E2 -2961.87} C_VEL
LIN {X 0,Y 558.943,Z 614.624,A -85,B 0,C 180,E1 -2962.959,E2 -2962.959} C_VEL
LIN {X 0,Y 558.935,Z 621.681,A -85,B 0,C 180,E1 -2964.227,E2 -2964.227} C_VEL
LIN {X 0,Y 558.827,Z 626.374,A -85,B 0,C 180,E1 -2965.311,E2 -2965.311} C_VEL
LIN {X 0,Y 558.836,Z 629.959,A -85,B 0,C 180,E1 -2966.395,E2 -2966.395} C_VEL
LIN {X 0,Y 558.799,Z 631.808,A -85,B 0,C 180,E1 -2967.117,E2 -2967.117} C_VEL
LIN {X 0,Y 558.745,Z 634.185,A -85,B 0,C 180,E1 -2968.559,E2 -2968.559} C_VEL
LIN {X 0,Y 558.74,Z 635,A -85,B 0,C 180,E1 -2970,E2 -2970} C_VEL
LIN {X 0,Y 558.745,Z 634.185,A -85,B 0,C 180,E1 -2971.442,E2 -2971.442} C_VEL
LIN {X 0,Y 558.799,Z 631.81,A -85,B 0,C 180,E1 -2972.884,E2 -2972.884} C_VEL
LIN {X 0,Y 558.844,Z 628.895,A -85,B 0,C 180,E1 -2973.966,E2 -2973.966} C_VEL
LIN {X 0,Y 558.799,Z 624.948,A -85,B 0,C 180,E1 -2975.051,E2 -2975.051} C_VEL
LIN {X 0,Y 558.921,Z 619.867,A -85,B 0,C 180,E1 -2976.136,E2 -2976.136} C_VEL
LIN {X 0,Y 558.977,Z 613.467,A -85,B 0,C 180,E1 -2977.223,E2 -2977.223} C_VEL
LIN {X 0,Y 559.099,Z 605.478,A -85,B 0,C 180,E1 -2978.312,E2 -2978.312} C_VEL
LIN {X 0,Y 559.184,Z 597.335,A -85,B 0,C 180,E1 -2979.221,E2 -2979.221} C_VEL
LIN {X 0,Y 559.351,Z 587.4,A -85,B 0,C 180,E1 -2980.131,E2 -2980.131} C_VEL
LIN {X 0,Y 559.53,Z 576.366,A -85,B 0,C 180,E1 -2980.939,E2 -2980.939} C_VEL
LIN {X 0,Y 559.704,Z 564.142,A -85,B 0,C 180,E1 -2981.644,E2 -2981.644} C_VEL
LIN {X 0,Y 559.833,Z 551.769,A -85,B 0,C 180,E1 -2982.184,E2 -2982.184} C_VEL
LIN {X 0,Y 559.965,Z 538.349,A -85,B 0,C 180,E1 -2982.596,E2 -2982.596} C_VEL
LIN {X 0,Y 560.097,Z 525.09,A -85,B 0,C 180,E1 -2982.846,E2 -2982.846} C_VEL
LIN {X 0,Y 560.186,Z 428.765,A -85,B 0,C 180,E1 -2984.088,E2 -2984.088} C_VEL
LIN {X 0,Y 559.379,Z 423.304,A -85,B 0,C 180,E1 -2984.205,E2 -2984.205} C_VEL
LIN {X 0,Y 559.564,Z 404.551,A -85,B 0,C 180,E1 -2987.068,E2 -2987.068} C_VEL
LIN {X 0,Y 559.85,Z 384.552,A -85,B 0,C 180,E1 -2990.195,E2 -2990.195} C_VEL
LIN {X 0,Y 559.98,Z 373.862,A -85,B 0,C 180,E1 -2991.888,E2 -2991.888} C_VEL
LIN {X 0,Y 559.182,Z 369.429,A -85,B 0,C 180,E1 -2992.662,E2 -2992.662} C_VEL
LIN {X 0,Y 559.178,Z 369.334,A -85,B 0,C 180,E1 -2995.298,E2 -2995.298} C_VEL
LIN {X 0,Y 559.183,Z 369.333,A -85,B 0,C 180,E1 -2997.712,E2 -2997.712} C_VEL
LIN {X 0,Y 559.158,Z 369.329,A -85,B 0,C 180,E1 -3000.182,E2 -3000.182} C_VEL
LIN {X 0,Y 559.176,Z 369.327,A -85,B 0,C 180,E1 -3002.713,E2 -3002.713} C_VEL
LIN {X 0,Y 559.16,Z 369.337,A -85,B 0,C 180,E1 -3005.321,E2 -3005.321} C_VEL
LIN {X 0,Y 559.135,Z 369.333,A -85,B 0,C 180,E1 -3008.017,E2 -3008.017} C_VEL
LIN {X 0,Y 559.176,Z 369.33,A -85,B 0,C 180,E1 -3010.81,E2 -3010.81} C_VEL
LIN {X 0,Y 559.161,Z 369.331,A -85,B 0,C 180,E1 -3013.731,E2 -3013.731} C_VEL
LIN {X 0,Y 559.169,Z 369.332,A -85,B 0,C 180,E1 -3016.8,E2 -3016.8} C_VEL
LIN {X 0,Y 559.178,Z 369.335,A -85,B 0,C 180,E1 -3019.189,E2 -3019.189} C_VEL
LIN {X 0,Y 559.133,Z 369.332,A -85,B 0,C 180,E1 -3021.982,E2 -3021.982} C_VEL
LIN {X 0,Y 559.156,Z 369.335,A -85,B 0,C 180,E1 -3024.782,E2 -3024.782} C_VEL
LIN {X 0,Y 559.171,Z 369.331,A -85,B 0,C 180,E1 -3027.361,E2 -3027.361} C_VEL
LIN {X 0,Y 559.145,Z 369.331,A -85,B 0,C 180,E1 -3030.142,E2 -3030.142} C_VEL
LIN {X 0,Y 559.177,Z 369.332,A -85,B 0,C 180,E1 -3033.169,E2 -3033.169} C_VEL
LIN {X 0,Y 559.151,Z 369.331,A -85,B 0,C 180,E1 -3035.494,E2 -3035.494} C_VEL
LIN {X 0,Y 559.172,Z 369.335,A -85,B 0,C 180,E1 -3038.624,E2 -3038.624} C_VEL
LIN {X 0,Y 559.166,Z 369.335,A -85,B 0,C 180,E1 -3040.926,E2 -3040.926} C_VEL
LIN {X 0,Y 559.165,Z 369.329,A -85,B 0,C 180,E1 -3043.948,E2 -3043.948} C_VEL
LIN {X 0,Y 559.167,Z 369.331,A -85,B 0,C 180,E1 -3046.184,E2 -3046.184} C_VEL
LIN {X 0,Y 559.189,Z 369.328,A -85,B 0,C 180,E1 -3049.133,E2 -3049.133} C_VEL
LIN {X 0,Y 559.201,Z 369.327,A -85,B 0,C 180,E1 -3052.053,E2 -3052.053} C_VEL
LIN {X 0,Y 559.251,Z 369.321,A -85,B 0,C 180,E1 -3054.953,E2 -3054.953} C_VEL
LIN {X 0,Y 559.245,Z 369.321,A -85,B 0,C 180,E1 -3057.839,E2 -3057.839} C_VEL
LIN {X 0,Y 559.269,Z 369.32,A -85,B 0,C 180,E1 -3060.72,E2 -3060.72} C_VEL
LIN {X 0,Y 559.237,Z 369.322,A -85,B 0,C 180,E1 -3062.881,E2 -3062.881} C_VEL
LIN {X 0,Y 559.224,Z 369.324,A -85,B 0,C 180,E1 -3065.77,E2 -3065.77} C_VEL
LIN {X 0,Y 559.186,Z 369.329,A -85,B 0,C 180,E1 -3068.674,E2 -3068.674} C_VEL
LIN {X 0,Y 559.198,Z 369.326,A -85,B 0,C 180,E1 -3071.601,E2 -3071.601} C_VEL
LIN {X 0,Y 559.193,Z 369.328,A -85,B 0,C 180,E1 -3074.596,E2 -3074.596} C_VEL
LIN {X 0,Y 559.159,Z 369.332,A -85,B 0,C 180,E1 -3077.557,E2 -3077.557} C_VEL
LIN {X 0,Y 559.169,Z 369.335,A -85,B 0,C 180,E1 -3079.837,E2 -3079.837} C_VEL
LIN {X 0,Y 559.138,Z 369.339,A -85,B 0,C 180,E1 -3082.153,E2 -3082.153} C_VEL
LIN {X 0,Y 559.174,Z 369.328,A -85,B 0,C 180,E1 -3085.188,E2 -3085.188} C_VEL
LIN {X 0,Y 559.19,Z 369.333,A -85,B 0,C 180,E1 -3087.712,E2 -3087.712} C_VEL
LIN {X 0,Y 559.148,Z 369.331,A -85,B 0,C 180,E1 -3090.628,E2 -3090.628} C_VEL
LIN {X 0,Y 558.486,Z 369.416,A -85,B 0,C 180,E1 -3091.23,E2 -3091.23} C_VEL
LIN {X 0,Y 555.623,Z 369.773,A -85,B 0,C 180,E1 -3092.206,E2 -3092.206} C_VEL
LIN {X 0,Y 553.212,Z 370.072,A -85,B 0,C 180,E1 -3092.992,E2 -3092.992} C_VEL
LIN {X 0,Y 552.193,Z 370.204,A -85,B 0,C 180,E1 -3093.598,E2 -3093.598} C_VEL
LIN {X 0,Y 552.119,Z 370.209,A -85,B 0,C 180,E1 -3093.804,E2 -3093.804} C_VEL
LIN {X 0,Y 552.108,Z 370.208,A -85,B 0,C 180,E1 -3096.747,E2 -3096.747} C_VEL
LIN {X 0,Y 552.131,Z 370.212,A -85,B 0,C 180,E1 -3099.527,E2 -3099.527} C_VEL
LIN {X 0,Y 552.128,Z 370.206,A -85,B 0,C 180,E1 -3102.426,E2 -3102.426} C_VEL
LIN {X 0,Y 552.095,Z 370.217,A -85,B 0,C 180,E1 -3105.563,E2 -3105.563} C_VEL
LIN {X 0,Y 552.139,Z 370.204,A -85,B 0,C 180,E1 -3108.677,E2 -3108.677} C_VEL
LIN {X 0,Y 552.119,Z 370.215,A -85,B 0,C 180,E1 -3111.412,E2 -3111.412} C_VEL
LIN {X 0,Y 552.113,Z 370.207,A -85,B 0,C 180,E1 -3114.159,E2 -3114.159} C_VEL
LIN {X 0,Y 552.123,Z 370.208,A -85,B 0,C 180,E1 -3116.815,E2 -3116.815} C_VEL
LIN {X 0,Y 552.105,Z 370.215,A -85,B 0,C 180,E1 -3119.391,E2 -3119.391} C_VEL
LIN {X 0,Y 552.11,Z 370.208,A -85,B 0,C 180,E1 -3121.902,E2 -3121.902} C_VEL
LIN {X 0,Y 552.156,Z 370.203,A -85,B 0,C 180,E1 -3124.65,E2 -3124.65} C_VEL
LIN {X 0,Y 552.093,Z 370.213,A -85,B 0,C 180,E1 -3127.549,E2 -3127.549} C_VEL
LIN {X 0,Y 552.146,Z 370.203,A -85,B 0,C 180,E1 -3130.375,E2 -3130.375} C_VEL
LIN {X 0,Y 552.157,Z 370.209,A -85,B 0,C 180,E1 -3132.978,E2 -3132.978} C_VEL
LIN {X 0,Y 552.138,Z 370.204,A -85,B 0,C 180,E1 -3136.005,E2 -3136.005} C_VEL
LIN {X 0,Y 552.165,Z 370.209,A -85,B 0,C 180,E1 -3138.994,E2 -3138.994} C_VEL
LIN {X 0,Y 552.173,Z 370.381,A -85,B 0,C 180,E1 -3141.952,E2 -3141.952} C_VEL
LIN {X 0,Y 552.763,Z 375.801,A -85,B 0,C 180,E1 -3142.95,E2 -3142.95} C_VEL
LIN {X 0,Y 552.543,Z 390.009,A -85,B 0,C 180,E1 -3145.44,E2 -3145.44} C_VEL
LIN {X 0,Y 552.311,Z 408.017,A -85,B 0,C 180,E1 -3148.542,E2 -3148.542} C_VEL
LIN {X 0,Y 552.344,Z 409.245,A -85,B 0,C 180,E1 -3148.678,E2 -3148.678} C_VEL
LIN {X 0,Y 553.425,Z 416.516,A -85,B 0,C 180,E1 -3148.817,E2 -3148.817} C_VEL
LIN {X 0,Y 553.124,Z 516.371,A -85,B 0,C 180,E1 -3150.136,E2 -3150.136} C_VEL
LIN {X 0,Y 553.026,Z 530.05,A -85,B 0,C 180,E1 -3150.478,E2 -3150.478} C_VEL
LIN {X 0,Y 552.819,Z 542.921,A -85,B 0,C 180,E1 -3150.956,E2 -3150.956} C_VEL
LIN {X 0,Y 552.598,Z 554.621,A -85,B 0,C 180,E1 -3151.548,E2 -3151.548} C_VEL
LIN {X 0,Y 552.448,Z 565.87,A -85,B 0,C 180,E1 -3152.278,E2 -3152.278} C_VEL
LIN {X 0,Y 552.248,Z 576.066,A -85,B 0,C 180,E1 -3153.1,E2 -3153.1} C_VEL
LIN {X 0,Y 552.063,Z 585.27,A -85,B 0,C 180,E1 -3154.015,E2 -3154.015} C_VEL
LIN {X 0,Y 551.921,Z 594.22,A -85,B 0,C 180,E1 -3155.114,E2 -3155.114} C_VEL
LIN {X 0,Y 551.869,Z 600.731,A -85,B 0,C 180,E1 -3156.095,E2 -3156.095} C_VEL
LIN {X 0,Y 551.803,Z 607.268,A -85,B 0,C 180,E1 -3157.317,E2 -3157.317} C_VEL
LIN {X 0,Y 551.748,Z 611.859,A -85,B 0,C 180,E1 -3158.423,E2 -3158.423} C_VEL
LIN {X 0,Y 551.688,Z 615.361,A -85,B 0,C 180,E1 -3159.532,E2 -3159.532} C_VEL
LIN {X 0,Y 551.679,Z 617.113,A -85,B 0,C 180,E1 -3160.273,E2 -3160.273} C_VEL
LIN {X 0,Y 551.71,Z 618.762,A -85,B 0,C 180,E1 -3161.224,E2 -3161.224} C_VEL
LIN {X 0,Y 551.657,Z 619.889,A -85,B 0,C 180,E1 -3162.508,E2 -3162.508} C_VEL
LIN {X 0,Y 551.656,Z 619.961,A -85,B 0,C 180,E1 -3163.256,E2 -3163.256} C_VEL
LIN {X 0,Y 551.694,Z 619.192,A -85,B 0,C 180,E1 -3164.497,E2 -3164.497} C_VEL
LIN {X 0,Y 551.619,Z 617.703,A -85,B 0,C 180,E1 -3165.518,E2 -3165.518} C_VEL
LIN {X 0,Y 551.702,Z 615.078,A -85,B 0,C 180,E1 -3166.655,E2 -3166.655} C_VEL
LIN {X 0,Y 551.737,Z 611.349,A -85,B 0,C 180,E1 -3167.8,E2 -3167.8} C_VEL
LIN {X 0,Y 551.82,Z 606.393,A -85,B 0,C 180,E1 -3168.951,E2 -3168.951} C_VEL
LIN {X 0,Y 551.874,Z 600.03,A -85,B 0,C 180,E1 -3170.11,E2 -3170.11} C_VEL
LIN {X 0,Y 552.008,Z 592,A -85,B 0,C 180,E1 -3171.275,E2 -3171.275} C_VEL
LIN {X 0,Y 552.121,Z 583.618,A -85,B 0,C 180,E1 -3172.252,E2 -3172.252} C_VEL
LIN {X 0,Y 552.323,Z 573.267,A -85,B 0,C 180,E1 -3173.231,E2 -3173.231} C_VEL
LIN {X 0,Y 552.496,Z 562.965,A -85,B 0,C 180,E1 -3174.019,E2 -3174.019} C_VEL
LIN {X 0,Y 552.677,Z 551.571,A -85,B 0,C 180,E1 -3174.711,E2 -3174.711} C_VEL
LIN {X 0,Y 552.867,Z 540.292,A -85,B 0,C 180,E1 -3175.243,E2 -3175.243} C_VEL
LIN {X 0,Y 553.053,Z 527.222,A -85,B 0,C 180,E1 -3175.699,E2 -3175.699} C_VEL
LIN {X 0,Y 553.114,Z 515.376,A -85,B 0,C 180,E1 -3175.974,E2 -3175.974} C_VEL
LIN {X 0,Y 553.373,Z 415.868,A -85,B 0,C 180,E1 -3177.282,E2 -3177.282} C_VEL
LIN {X 0,Y 552.265,Z 409.135,A -85,B 0,C 180,E1 -3177.419,E2 -3177.419} C_VEL
LIN {X 0,Y 552.244,Z 407.266,A -85,B 0,C 180,E1 -3177.677,E2 -3177.677} C_VEL
LIN {X 0,Y 552.482,Z 390.406,A -85,B 0,C 180,E1 -3180.585,E2 -3180.585} C_VEL
LIN {X 0,Y 552.785,Z 374.578,A -85,B 0,C 180,E1 -3183.357,E2 -3183.357} C_VEL
LIN {X 0,Y 552.148,Z 370.294,A -85,B 0,C 180,E1 -3184.172,E2 -3184.172} C_VEL
LIN {X 0,Y 552.115,Z 370.212,A -85,B 0,C 180,E1 -3186.745,E2 -3186.745} C_VEL
LIN {X 0,Y 552.131,Z 370.209,A -85,B 0,C 180,E1 -3189.526,E2 -3189.526} C_VEL
LIN {X 0,Y 552.126,Z 370.206,A -85,B 0,C 180,E1 -3192.425,E2 -3192.425} C_VEL
LIN {X 0,Y 552.095,Z 370.212,A -85,B 0,C 180,E1 -3195.562,E2 -3195.562} C_VEL
LIN {X 0,Y 552.166,Z 370.201,A -85,B 0,C 180,E1 -3198.672,E2 -3198.672} C_VEL
LIN {X 0,Y 552.115,Z 370.21,A -85,B 0,C 180,E1 -3201.411,E2 -3201.411} C_VEL
LIN {X 0,Y 552.107,Z 370.207,A -85,B 0,C 180,E1 -3204.158,E2 -3204.158} C_VEL
LIN {X 0,Y 552.122,Z 370.21,A -85,B 0,C 180,E1 -3206.815,E2 -3206.815} C_VEL
LIN {X 0,Y 552.108,Z 370.207,A -85,B 0,C 180,E1 -3209.391,E2 -3209.391} C_VEL
LIN {X 0,Y 552.12,Z 370.205,A -85,B 0,C 180,E1 -3211.902,E2 -3211.902} C_VEL
LIN {X 0,Y 552.148,Z 370.206,A -85,B 0,C 180,E1 -3214.649,E2 -3214.649} C_VEL
LIN {X 0,Y 552.107,Z 370.207,A -85,B 0,C 180,E1 -3217.55,E2 -3217.55} C_VEL
LIN {X 0,Y 552.155,Z 370.206,A -85,B 0,C 180,E1 -3220.674,E2 -3220.674} C_VEL
LIN {X 0,Y 552.115,Z 370.206,A -85,B 0,C 180,E1 -3223.737,E2 -3223.737} C_VEL
LIN {X 0,Y 552.129,Z 370.203,A -85,B 0,C 180,E1 -3226.004,E2 -3226.004} C_VEL
LIN {X 0,Y 552.17,Z 370.205,A -85,B 0,C 180,E1 -3228.994,E2 -3228.994} C_VEL
LIN {X 0,Y 552.158,Z 370.2,A -85,B 0,C 180,E1 -3231.952,E2 -3231.952} C_VEL
LIN {X 0,Y 552.226,Z 370.2,A -85,B 0,C 180,E1 -3234.889,E2 -3234.889} C_VEL
LIN {X 0,Y 552.216,Z 370.193,A -85,B 0,C 180,E1 -3237.812,E2 -3237.812} C_VEL
LIN {X 0,Y 552.241,Z 370.197,A -85,B 0,C 180,E1 -3240.729,E2 -3240.729} C_VEL
LIN {X 0,Y 552.205,Z 370.2,A -85,B 0,C 180,E1 -3242.918,E2 -3242.918} C_VEL
LIN {X 0,Y 552.193,Z 370.196,A -85,B 0,C 180,E1 -3245.844,E2 -3245.844} C_VEL
LIN {X 0,Y 552.164,Z 370.207,A -85,B 0,C 180,E1 -3248.786,E2 -3248.786} C_VEL
LIN {X 0,Y 552.155,Z 370.201,A -85,B 0,C 180,E1 -3251.751,E2 -3251.751} C_VEL
LIN {X 0,Y 552.128,Z 370.212,A -85,B 0,C 180,E1 -3254.749,E2 -3254.749} C_VEL
LIN {X 0,Y 552.108,Z 370.205,A -85,B 0,C 180,E1 -3257.789,E2 -3257.789} C_VEL
LIN {X 0,Y 552.127,Z 370.206,A -85,B 0,C 180,E1 -3260.101,E2 -3260.101} C_VEL
LIN {X 0,Y 552.107,Z 370.212,A -85,B 0,C 180,E1 -3262.45,E2 -3262.45} C_VEL
LIN {X 0,Y 552.149,Z 370.202,A -85,B 0,C 180,E1 -3265.351,E2 -3265.351} C_VEL
LIN {X 0,Y 552.12,Z 370.207,A -85,B 0,C 180,E1 -3268.098,E2 -3268.098} C_VEL
LIN {X 0,Y 552.101,Z 370.216,A -85,B 0,C 180,E1 -3270.61,E2 -3270.61} C_VEL
LIN {X 0,Y 552.123,Z 370.206,A -85,B 0,C 180,E1 -3273.186,E2 -3273.186} C_VEL
LIN {X 0,Y 552.107,Z 370.207,A -85,B 0,C 180,E1 -3275.842,E2 -3275.842} C_VEL
LIN {X 0,Y 552.121,Z 370.208,A -85,B 0,C 180,E1 -3279.063,E2 -3279.063} C_VEL
LIN {X 0,Y 552.14,Z 370.199,A -85,B 0,C 180,E1 -3281.444,E2 -3281.444} C_VEL
LIN {X 0,Y 552.093,Z 370.218,A -85,B 0,C 180,E1 -3284.533,E2 -3284.533} C_VEL
LIN {X 0,Y 552.127,Z 370.204,A -85,B 0,C 180,E1 -3287.585,E2 -3287.585} C_VEL
LIN {X 0,Y 552.132,Z 370.211,A -85,B 0,C 180,E1 -3290.474,E2 -3290.474} C_VEL
LIN {X 0,Y 552.113,Z 370.205,A -85,B 0,C 180,E1 -3293.316,E2 -3293.316} C_VEL
LIN {X 0,Y 552.139,Z 370.205,A -85,B 0,C 180,E1 -3295.941,E2 -3295.941} C_VEL
LIN {X 0,Y 552.118,Z 370.214,A -85,B 0,C 180,E1 -3298.541,E2 -3298.541} C_VEL
LIN {X 0,Y 552.124,Z 370.206,A -85,B 0,C 180,E1 -3301.439,E2 -3301.439} C_VEL
LIN {X 0,Y 552.138,Z 370.212,A -85,B 0,C 180,E1 -3304.357,E2 -3304.357} C_VEL
LIN {X 0,Y 552.144,Z 370.342,A -85,B 0,C 180,E1 -3307.206,E2 -3307.206} C_VEL
LIN {X 0,Y 553.016,Z 375.387,A -85,B 0,C 180,E1 -3308.083,E2 -3308.083} C_VEL
LIN {X 0,Y 552.796,Z 390.103,A -85,B 0,C 180,E1 -3310.436,E2 -3310.436} C_VEL
LIN {X 0,Y 552.552,Z 406.314,A -85,B 0,C 180,E1 -3312.99,E2 -3312.99} C_VEL
LIN {X 0,Y 552.404,Z 423.325,A -85,B 0,C 180,E1 -3315.613,E2 -3315.613} C_VEL
LIN {X 0,Y 553.431,Z 430.995,A -85,B 0,C 180,E1 -3315.766,E2 -3315.766} C_VEL
LIN {X 0,Y 553.164,Z 530.968,A -85,B 0,C 180,E1 -3317.084,E2 -3317.084} C_VEL
LIN {X 0,Y 553.016,Z 544.232,A -85,B 0,C 180,E1 -3317.407,E2 -3317.407} C_VEL
LIN {X 0,Y 552.848,Z 556.38,A -85,B 0,C 180,E1 -3317.846,E2 -3317.846} C_VEL
LIN {X 0,Y 552.69,Z 568.668,A -85,B 0,C 180,E1 -3318.449,E2 -3318.449} C_VEL
LIN {X 0,Y 552.487,Z 580.201,A -85,B 0,C 180,E1 -3319.186,E2 -3319.186} C_VEL
LIN {X 0,Y 552.272,Z 590.609,A -85,B 0,C 180,E1 -3320.016,E2 -3320.016} C_VEL
LIN {X 0,Y 552.125,Z 599.117,A -85,B 0,C 180,E1 -3320.845,E2 -3320.845} C_VEL
LIN {X 0,Y 552.013,Z 606.963,A -85,B 0,C 180,E1 -3321.766,E2 -3321.766} C_VEL
LIN {X 0,Y 551.889,Z 614.624,A -85,B 0,C 180,E1 -3322.868,E2 -3322.868} C_VEL
LIN {X 0,Y 551.867,Z 621.681,A -85,B 0,C 180,E1 -3324.153,E2 -3324.153} C_VEL
LIN {X 0,Y 551.725,Z 626.374,A -85,B 0,C 180,E1 -3325.251,E2 -3325.251} C_VEL
LIN {X 0,Y 551.75,Z 629.959,A -85,B 0,C 180,E1 -3326.349,E2 -3326.349} C_VEL
LIN {X 0,Y 551.724,Z 631.808,A -85,B 0,C 180,E1 -3327.08,E2 -3327.08} C_VEL
LIN {X 0,Y 551.645,Z 634.184,A -85,B 0,C 180,E1 -3328.54,E2 -3328.54} C_VEL
LIN {X 0,Y 551.64,Z 635,A -85,B 0,C 180,E1 -3330,E2 -3330} C_VEL
LIN {X 0,Y 551.645,Z 634.185,A -85,B 0,C 180,E1 -3331.46,E2 -3331.46} C_VEL
LIN {X 0,Y 551.724,Z 631.81,A -85,B 0,C 180,E1 -3332.921,E2 -3332.921} C_VEL
LIN {X 0,Y 551.764,Z 628.895,A -85,B 0,C 180,E1 -3334.017,E2 -3334.017} C_VEL
LIN {X 0,Y 551.724,Z 624.948,A -85,B 0,C 180,E1 -3335.116,E2 -3335.116} C_VEL
LIN {X 0,Y 551.815,Z 619.124,A -85,B 0,C 180,E1 -3336.353,E2 -3336.353} C_VEL
LIN {X 0,Y 551.926,Z 612.236,A -85,B 0,C 180,E1 -3337.5,E2 -3337.5} C_VEL
LIN {X 0,Y 552.082,Z 603.991,A -85,B 0,C 180,E1 -3338.602,E2 -3338.602} C_VEL
LIN {X 0,Y 552.221,Z 595.539,A -85,B 0,C 180,E1 -3339.523,E2 -3339.523} C_VEL
LIN {X 0,Y 552.411,Z 585.094,A -85,B 0,C 180,E1 -3340.445,E2 -3340.445} C_VEL
LIN {X 0,Y 552.583,Z 574.129,A -85,B 0,C 180,E1 -3341.224,E2 -3341.224} C_VEL
LIN {X 0,Y 552.784,Z 563.407,A -85,B 0,C 180,E1 -3341.83,E2 -3341.83} C_VEL
LIN {X 0,Y 552.912,Z 551.766,A -85,B 0,C 180,E1 -3342.339,E2 -3342.339} C_VEL
LIN {X 0,Y 553.04,Z 538.348,A -85,B 0,C 180,E1 -3342.756,E2 -3342.756} C_VEL
LIN {X 0,Y 553.177,Z 525.09,A -85,B 0,C 180,E1 -3343.009,E2 -3343.009} C_VEL
LIN {X 0,Y 553.337,Z 429.681,A -85,B 0,C 180,E1 -3344.254,E2 -3344.254} C_VEL
LIN {X 0,Y 552.385,Z 423.329,A -85,B 0,C 180,E1 -3344.387,E2 -3344.387} C_VEL
LIN {X 0,Y 552.669,Z 401.456,A -85,B 0,C 180,E1 -3347.77,E2 -3347.77} C_VEL
LIN {X 0,Y 553.005,Z 379.624,A -85,B 0,C 180,E1 -3351.235,E2 -3351.235} C_VEL
LIN {X 0,Y 552.872,Z 374.198,A -85,B 0,C 180,E1 -3352.118,E2 -3352.118} C_VEL
LIN {X 0,Y 552.138,Z 370.289,A -85,B 0,C 180,E1 -3352.819,E2 -3352.819} C_VEL
LIN {X 0,Y 552.133,Z 370.213,A -85,B 0,C 180,E1 -3355.644,E2 -3355.644} C_VEL
LIN {X 0,Y 552.126,Z 370.206,A -85,B 0,C 180,E1 -3358.562,E2 -3358.562} C_VEL
LIN {X 0,Y 552.137,Z 370.213,A -85,B 0,C 180,E1 -3361.479,E2 -3361.479} C_VEL
LIN {X 0,Y 552.139,Z 370.203,A -85,B 0,C 180,E1 -3364.171,E2 -3364.171} C_VEL
LIN {X 0,Y 552.112,Z 370.208,A -85,B 0,C 180,E1 -3366.746,E2 -3366.746} C_VEL
LIN {X 0,Y 552.134,Z 370.21,A -85,B 0,C 180,E1 -3369.526,E2 -3369.526} C_VEL
LIN {X 0,Y 552.129,Z 370.205,A -85,B 0,C 180,E1 -3372.425,E2 -3372.425} C_VEL
LIN {X 0,Y 552.098,Z 370.212,A -85,B 0,C 180,E1 -3375.562,E2 -3375.562} C_VEL
LIN {X 0,Y 552.169,Z 370.203,A -85,B 0,C 180,E1 -3378.672,E2 -3378.672} C_VEL
LIN {X 0,Y 552.118,Z 370.211,A -85,B 0,C 180,E1 -3381.411,E2 -3381.411} C_VEL
LIN {X 0,Y 552.11,Z 370.207,A -85,B 0,C 180,E1 -3384.158,E2 -3384.158} C_VEL
LIN {X 0,Y 552.119,Z 370.212,A -85,B 0,C 180,E1 -3386.814,E2 -3386.814} C_VEL
LIN {X 0,Y 552.103,Z 370.211,A -85,B 0,C 180,E1 -3389.391,E2 -3389.391} C_VEL
LIN {X 0,Y 552.122,Z 370.206,A -85,B 0,C 180,E1 -3391.902,E2 -3391.902} C_VEL
LIN {X 0,Y 552.152,Z 370.208,A -85,B 0,C 180,E1 -3394.649,E2 -3394.649} C_VEL
LIN {X 0,Y 552.091,Z 370.21,A -85,B 0,C 180,E1 -3397.549,E2 -3397.549} C_VEL
LIN {X 0,Y 552.144,Z 370.207,A -85,B 0,C 180,E1 -3400.373,E2 -3400.373} C_VEL
LIN {X 0,Y 552.152,Z 370.207,A -85,B 0,C 180,E1 -3402.977,E2 -3402.977} C_VEL
LIN {X 0,Y 552.13,Z 370.206,A -85,B 0,C 180,E1 -3406.004,E2 -3406.004} C_VEL
LIN {X 0,Y 552.156,Z 370.205,A -85,B 0,C 180,E1 -3408.993,E2 -3408.993} C_VEL
LIN {X 0,Y 552.154,Z 370.204,A -85,B 0,C 180,E1 -3411.951,E2 -3411.951} C_VEL
LIN {X 0,Y 552.226,Z 370.197,A -85,B 0,C 180,E1 -3414.889,E2 -3414.889} C_VEL
LIN {X 0,Y 552.217,Z 370.196,A -85,B 0,C 180,E1 -3417.812,E2 -3417.812} C_VEL
LIN {X 0,Y 552.239,Z 370.196,A -85,B 0,C 180,E1 -3420.729,E2 -3420.729} C_VEL
LIN {X 0,Y 552.204,Z 370.198,A -85,B 0,C 180,E1 -3422.918,E2 -3422.918} C_VEL
LIN {X 0,Y 552.194,Z 370.201,A -85,B 0,C 180,E1 -3425.844,E2 -3425.844} C_VEL
LIN {X 0,Y 552.156,Z 370.204,A -85,B 0,C 180,E1 -3428.786,E2 -3428.786} C_VEL
LIN {X 0,Y 552.156,Z 370.205,A -85,B 0,C 180,E1 -3431.751,E2 -3431.751} C_VEL
LIN {X 0,Y 552.131,Z 370.207,A -85,B 0,C 180,E1 -3434.749,E2 -3434.749} C_VEL
LIN {X 0,Y 552.11,Z 370.213,A -85,B 0,C 180,E1 -3437.788,E2 -3437.788} C_VEL
LIN {X 0,Y 552.129,Z 370.212,A -85,B 0,C 180,E1 -3440.101,E2 -3440.101} C_VEL
LIN {X 0,Y 552.092,Z 370.213,A -85,B 0,C 180,E1 -3442.451,E2 -3442.451} C_VEL
LIN {X 0,Y 552.151,Z 370.204,A -85,B 0,C 180,E1 -3445.351,E2 -3445.351} C_VEL
LIN {X 0,Y 552.122,Z 370.212,A -85,B 0,C 180,E1 -3448.098,E2 -3448.098} C_VEL
LIN {X 0,Y 552.109,Z 370.208,A -85,B 0,C 180,E1 -3450.623,E2 -3450.623} C_VEL
LIN {X 0,Y 552.125,Z 370.207,A -85,B 0,C 180,E1 -3453.185,E2 -3453.185} C_VEL
LIN {X 0,Y 552.119,Z 370.209,A -85,B 0,C 180,E1 -3453.804,E2 -3453.804} C_VEL
LIN {X 0,Y 551.484,Z 370.291,A -85,B 0,C 180,E1 -3454.412,E2 -3454.412} C_VEL
LIN {X 0,Y 548.658,Z 370.642,A -85,B 0,C 180,E1 -3455.4,E2 -3455.4} C_VEL
LIN {X 0,Y 546.233,Z 370.943,A -85,B 0,C 180,E1 -3456.196,E2 -3456.196} C_VEL
LIN {X 0,Y 545.163,Z 371.073,A -85,B 0,C 180,E1 -3456.809,E2 -3456.809} C_VEL
LIN {X 0,Y 545.061,Z 371.087,A -85,B 0,C 180,E1 -3457.017,E2 -3457.017} C_VEL
LIN {X 0,Y 545.072,Z 371.087,A -85,B 0,C 180,E1 -3460.142,E2 -3460.142} C_VEL
LIN {X 0,Y 545.084,Z 371.085,A -85,B 0,C 180,E1 -3463.106,E2 -3463.106} C_VEL
LIN {X 0,Y 545.064,Z 371.086,A -85,B 0,C 180,E1 -3466.225,E2 -3466.225} C_VEL
LIN {X 0,Y 545.1,Z 371.082,A -85,B 0,C 180,E1 -3468.888,E2 -3468.888} C_VEL
LIN {X 0,Y 545.053,Z 371.091,A -85,B 0,C 180,E1 -3471.763,E2 -3471.763} C_VEL
LIN {X 0,Y 545.065,Z 371.085,A -85,B 0,C 180,E1 -3474.534,E2 -3474.534} C_VEL
LIN {X 0,Y 545.081,Z 371.09,A -85,B 0,C 180,E1 -3477.213,E2 -3477.213} C_VEL
LIN {X 0,Y 545.065,Z 371.087,A -85,B 0,C 180,E1 -3479.811,E2 -3479.811} C_VEL
LIN {X 0,Y 545.081,Z 371.083,A -85,B 0,C 180,E1 -3482.344,E2 -3482.344} C_VEL
LIN {X 0,Y 545.118,Z 371.082,A -85,B 0,C 180,E1 -3484.821,E2 -3484.821} C_VEL
LIN {X 0,Y 545.04,Z 371.095,A -85,B 0,C 180,E1 -3487.243,E2 -3487.243} C_VEL
LIN {X 0,Y 545.118,Z 371.079,A -85,B 0,C 180,E1 -3490.415,E2 -3490.415} C_VEL
LIN {X 0,Y 545.073,Z 371.086,A -85,B 0,C 180,E1 -3493.521,E2 -3493.521} C_VEL
LIN {X 0,Y 545.097,Z 371.081,A -85,B 0,C 180,E1 -3495.82,E2 -3495.82} C_VEL
LIN {X 0,Y 545.121,Z 371.086,A -85,B 0,C 180,E1 -3498.849,E2 -3498.849} C_VEL
LIN {X 0,Y 545.135,Z 371.214,A -85,B 0,C 180,E1 -3501.8,E2 -3501.8} C_VEL
LIN {X 0,Y 545.806,Z 376.793,A -85,B 0,C 180,E1 -3502.847,E2 -3502.847} C_VEL
LIN {X 0,Y 545.543,Z 391.075,A -85,B 0,C 180,E1 -3505.382,E2 -3505.382} C_VEL
LIN {X 0,Y 545.303,Z 408.794,A -85,B 0,C 180,E1 -3508.454,E2 -3508.454} C_VEL
LIN {X 0,Y 545.596,Z 410.914,A -85,B 0,C 180,E1 -3508.534,E2 -3508.534} C_VEL
LIN {X 0,Y 546.569,Z 417.007,A -85,B 0,C 180,E1 -3508.641,E2 -3508.641} C_VEL
LIN {X 0,Y 546.198,Z 516.708,A -85,B 0,C 180,E1 -3509.977,E2 -3509.977} C_VEL
LIN {X 0,Y 546.087,Z 530.278,A -85,B 0,C 180,E1 -3510.322,E2 -3510.322} C_VEL
LIN {X 0,Y 545.86,Z 542.571,A -85,B 0,C 180,E1 -3510.784,E2 -3510.784} C_VEL
LIN {X 0,Y 545.651,Z 554.344,A -85,B 0,C 180,E1 -3511.384,E2 -3511.384} C_VEL
LIN {X 0,Y 545.443,Z 565.655,A -85,B 0,C 180,E1 -3512.123,E2 -3512.123} C_VEL
LIN {X 0,Y 545.211,Z 575.896,A -85,B 0,C 180,E1 -3512.955,E2 -3512.955} C_VEL
LIN {X 0,Y 545.02,Z 585.136,A -85,B 0,C 180,E1 -3513.882,E2 -3513.882} C_VEL
LIN {X 0,Y 544.885,Z 594.103,A -85,B 0,C 180,E1 -3514.994,E2 -3514.994} C_VEL
LIN {X 0,Y 544.782,Z 601.461,A -85,B 0,C 180,E1 -3516.126,E2 -3516.126} C_VEL
LIN {X 0,Y 544.701,Z 608.022,A -85,B 0,C 180,E1 -3517.413,E2 -3517.413} C_VEL
LIN {X 0,Y 544.668,Z 612.437,A -85,B 0,C 180,E1 -3518.533,E2 -3518.533} C_VEL
LIN {X 0,Y 544.605,Z 615.784,A -85,B 0,C 180,E1 -3519.657,E2 -3519.657} C_VEL
LIN {X 0,Y 544.582,Z 617.449,A -85,B 0,C 180,E1 -3520.409,E2 -3520.409} C_VEL
LIN {X 0,Y 544.62,Z 618.852,A -85,B 0,C 180,E1 -3521.264,E2 -3521.264} C_VEL
LIN {X 0,Y 544.567,Z 619.927,A -85,B 0,C 180,E1 -3522.673,E2 -3522.673} C_VEL
LIN {X 0,Y 544.555,Z 619.923,A -85,B 0,C 180,E1 -3523.432,E2 -3523.432} C_VEL
LIN {X 0,Y 544.591,Z 619.143,A -85,B 0,C 180,E1 -3524.56,E2 -3524.56} C_VEL
LIN {X 0,Y 544.549,Z 617.361,A -85,B 0,C 180,E1 -3525.725,E2 -3525.725} C_VEL
LIN {X 0,Y 544.635,Z 614.575,A -85,B 0,C 180,E1 -3526.878,E2 -3526.878} C_VEL
LIN {X 0,Y 544.674,Z 610.671,A -85,B 0,C 180,E1 -3528.039,E2 -3528.039} C_VEL
LIN {X 0,Y 544.741,Z 605.523,A -85,B 0,C 180,E1 -3529.207,E2 -3529.207} C_VEL
LIN {X 0,Y 544.811,Z 598.944,A -85,B 0,C 180,E1 -3530.383,E2 -3530.383} C_VEL
LIN {X 0,Y 544.969,Z 590.892,A -85,B 0,C 180,E1 -3531.522,E2 -3531.522} C_VEL
LIN {X 0,Y 545.131,Z 581.888,A -85,B 0,C 180,E1 -3532.553,E2 -3532.553} C_VEL
LIN {X 0,Y 545.317,Z 572.314,A -85,B 0,C 180,E1 -3533.447,E2 -3533.447} C_VEL
LIN {X 0,Y 545.503,Z 561.384,A -85,B 0,C 180,E1 -3534.268,E2 -3534.268} C_VEL
LIN {X 0,Y 545.76,Z 550.018,A -85,B 0,C 180,E1 -3534.944,E2 -3534.944} C_VEL
LIN {X 0,Y 545.949,Z 538.925,A -85,B 0,C 180,E1 -3535.458,E2 -3535.458} C_VEL
LIN {X 0,Y 546.124,Z 526.522,A -85,B 0,C 180,E1 -3535.883,E2 -3535.883} C_VEL
LIN {X 0,Y 546.225,Z 513.344,A -85,B 0,C 180,E1 -3536.172,E2 -3536.172} C_VEL
LIN {X 0,Y 546.489,Z 416.574,A -85,B 0,C 180,E1 -3537.457,E2 -3537.457} C_VEL
LIN {X 0,Y 545.266,Z 409.264,A -85,B 0,C 180,E1 -3537.603,E2 -3537.603} C_VEL
LIN {X 0,Y 545.26,Z 407.408,A -85,B 0,C 180,E1 -3537.854,E2 -3537.854} C_VEL
LIN {X 0,Y 545.531,Z 390.478,A -85,B 0,C 180,E1 -3540.821,E2 -3540.821} C_VEL
LIN {X 0,Y 545.826,Z 376.176,A -85,B 0,C 180,E1 -3543.355,E2 -3543.355} C_VEL
LIN {X 0,Y 545.09,Z 371.137,A -85,B 0,C 180,E1 -3544.329,E2 -3544.329} C_VEL
LIN {X 0,Y 545.067,Z 371.093,A -85,B 0,C 180,E1 -3547.3,E2 -3547.3} C_VEL
LIN {X 0,Y 545.089,Z 371.083,A -85,B 0,C 180,E1 -3550.139,E2 -3550.139} C_VEL
LIN {X 0,Y 545.082,Z 371.09,A -85,B 0,C 180,E1 -3553.105,E2 -3553.105} C_VEL
LIN {X 0,Y 545.062,Z 371.085,A -85,B 0,C 180,E1 -3556.223,E2 -3556.223} C_VEL
LIN {X 0,Y 545.118,Z 371.082,A -85,B 0,C 180,E1 -3558.889,E2 -3558.889} C_VEL
LIN {X 0,Y 545.049,Z 371.087,A -85,B 0,C 180,E1 -3561.762,E2 -3561.762} C_VEL
LIN {X 0,Y 545.059,Z 371.087,A -85,B 0,C 180,E1 -3564.533,E2 -3564.533} C_VEL
LIN {X 0,Y 545.076,Z 371.09,A -85,B 0,C 180,E1 -3567.212,E2 -3567.212} C_VEL
LIN {X 0,Y 545.094,Z 371.077,A -85,B 0,C 180,E1 -3569.812,E2 -3569.812} C_VEL
LIN {X 0,Y 545.095,Z 371.087,A -85,B 0,C 180,E1 -3572.824,E2 -3572.824} C_VEL
LIN {X 0,Y 545.051,Z 371.087,A -85,B 0,C 180,E1 -3575.631,E2 -3575.631} C_VEL
LIN {X 0,Y 545.072,Z 371.082,A -85,B 0,C 180,E1 -3578.175,E2 -3578.175} C_VEL
LIN {X 0,Y 545.113,Z 371.08,A -85,B 0,C 180,E1 -3580.415,E2 -3580.415} C_VEL
LIN {X 0,Y 545.07,Z 371.085,A -85,B 0,C 180,E1 -3583.521,E2 -3583.521} C_VEL
LIN {X 0,Y 545.087,Z 371.08,A -85,B 0,C 180,E1 -3585.82,E2 -3585.82} C_VEL
LIN {X 0,Y 545.124,Z 371.085,A -85,B 0,C 180,E1 -3588.85,E2 -3588.85} C_VEL
LIN {X 0,Y 545.128,Z 371.076,A -85,B 0,C 180,E1 -3591.847,E2 -3591.847} C_VEL
LIN {X 0,Y 545.201,Z 371.074,A -85,B 0,C 180,E1 -3594.823,E2 -3594.823} C_VEL
LIN {X 0,Y 545.187,Z 371.068,A -85,B 0,C 180,E1 -3597.784,E2 -3597.784} C_VEL
LIN {X 0,Y 545.211,Z 371.073,A -85,B 0,C 180,E1 -3600.739,E2 -3600.739} C_VEL
LIN {X 0,Y 545.171,Z 371.076,A -85,B 0,C 180,E1 -3602.956,E2 -3602.956} C_VEL
LIN {X 0,Y 545.164,Z 371.072,A -85,B 0,C 180,E1 -3605.92,E2 -3605.92} C_VEL
LIN {X 0,Y 545.12,Z 371.084,A -85,B 0,C 180,E1 -3608.9,E2 -3608.9} C_VEL
LIN {X 0,Y 545.127,Z 371.076,A -85,B 0,C 180,E1 -3611.904,E2 -3611.904} C_VEL
LIN {X 0,Y 545.077,Z 371.089,A -85,B 0,C 180,E1 -3614.944,E2 -3614.944} C_VEL
LIN {X 0,Y 545.076,Z 371.082,A -85,B 0,C 180,E1 -3618.026,E2 -3618.026} C_VEL
LIN {X 0,Y 545.091,Z 371.085,A -85,B 0,C 180,E1 -3620.372,E2 -3620.372} C_VEL
LIN {X 0,Y 545.106,Z 371.078,A -85,B 0,C 180,E1 -3623.558,E2 -3623.558} C_VEL
LIN {X 0,Y 545.082,Z 371.083,A -85,B 0,C 180,E1 -3626.001,E2 -3626.001} C_VEL
LIN {X 0,Y 545.084,Z 371.089,A -85,B 0,C 180,E1 -3628.749,E2 -3628.749} C_VEL
LIN {X 0,Y 545.071,Z 371.083,A -85,B 0,C 180,E1 -3631.683,E2 -3631.683} C_VEL
LIN {X 0,Y 545.078,Z 371.09,A -85,B 0,C 180,E1 -3634.563,E2 -3634.563} C_VEL
LIN {X 0,Y 545.036,Z 371.088,A -85,B 0,C 180,E1 -3637.304,E2 -3637.304} C_VEL
LIN {X 0,Y 545.089,Z 371.084,A -85,B 0,C 180,E1 -3640.141,E2 -3640.141} C_VEL
LIN {X 0,Y 545.084,Z 371.084,A -85,B 0,C 180,E1 -3643.106,E2 -3643.106} C_VEL
LIN {X 0,Y 545.061,Z 371.088,A -85,B 0,C 180,E1 -3646.225,E2 -3646.225} C_VEL
LIN {X 0,Y 545.094,Z 371.084,A -85,B 0,C 180,E1 -3648.888,E2 -3648.888} C_VEL
LIN {X 0,Y 545.052,Z 371.087,A -85,B 0,C 180,E1 -3651.764,E2 -3651.764} C_VEL
LIN {X 0,Y 545.065,Z 371.093,A -85,B 0,C 180,E1 -3654.535,E2 -3654.535} C_VEL
LIN {X 0,Y 545.082,Z 371.084,A -85,B 0,C 180,E1 -3657.213,E2 -3657.213} C_VEL
LIN {X 0,Y 545.066,Z 371.087,A -85,B 0,C 180,E1 -3659.812,E2 -3659.812} C_VEL
LIN {X 0,Y 545.094,Z 371.089,A -85,B 0,C 180,E1 -3662.345,E2 -3662.345} C_VEL
LIN {X 0,Y 545.119,Z 371.084,A -85,B 0,C 180,E1 -3664.821,E2 -3664.821} C_VEL
LIN {X 0,Y 545.106,Z 371.282,A -85,B 0,C 180,E1 -3667.071,E2 -3667.071} C_VEL
LIN {X 0,Y 546.06,Z 377.115,A -85,B 0,C 180,E1 -3668.085,E2 -3668.085} C_VEL
LIN {X 0,Y 545.799,Z 391.66,A -85,B 0,C 180,E1 -3670.441,E2 -3670.441} C_VEL
LIN {X 0,Y 545.538,Z 407.436,A -85,B 0,C 180,E1 -3672.958,E2 -3672.958} C_VEL
LIN {X 0,Y 545.379,Z 423.296,A -85,B 0,C 180,E1 -3675.424,E2 -3675.424} C_VEL
LIN {X 0,Y 546.553,Z 432.049,A -85,B 0,C 180,E1 -3675.597,E2 -3675.597} C_VEL
LIN {X 0,Y 546.248,Z 530.968,A -85,B 0,C 180,E1 -3676.918,E2 -3676.918} C_VEL
LIN {X 0,Y 546.103,Z 544.231,A -85,B 0,C 180,E1 -3677.245,E2 -3677.245} C_VEL
LIN {X 0,Y 545.9,Z 556.379,A -85,B 0,C 180,E1 -3677.689,E2 -3677.689} C_VEL
LIN {X 0,Y 545.731,Z 568.666,A -85,B 0,C 180,E1 -3678.3,E2 -3678.3} C_VEL
LIN {X 0,Y 545.506,Z 580.199,A -85,B 0,C 180,E1 -3679.046,E2 -3679.046} C_VEL
LIN {X 0,Y 545.261,Z 590.61,A -85,B 0,C 180,E1 -3679.886,E2 -3679.886} C_VEL
LIN {X 0,Y 545.084,Z 599.117,A -85,B 0,C 180,E1 -3680.726,E2 -3680.726} C_VEL
LIN {X 0,Y 544.977,Z 606.963,A -85,B 0,C 180,E1 -3681.658,E2 -3681.658} C_VEL
LIN {X 0,Y 544.823,Z 614.623,A -85,B 0,C 180,E1 -3682.775,E2 -3682.775} C_VEL
LIN {X 0,Y 544.776,Z 621.681,A -85,B 0,C 180,E1 -3684.077,E2 -3684.077} C_VEL
LIN {X 0,Y 544.629,Z 626.374,A -85,B 0,C 180,E1 -3685.189,E2 -3685.189} C_VEL
LIN {X 0,Y 544.669,Z 629.959,A -85,B 0,C 180,E1 -3686.301,E2 -3686.301} C_VEL
LIN {X 0,Y 544.65,Z 631.808,A -85,B 0,C 180,E1 -3687.042,E2 -3687.042} C_VEL
LIN {X 0,Y 544.546,Z 634.183,A -85,B 0,C 180,E1 -3688.521,E2 -3688.521} C_VEL
LIN {X 0,Y 544.541,Z 635,A -85,B 0,C 180,E1 -3690,E2 -3690} C_VEL
LIN {X 0,Y 544.546,Z 634.184,A -85,B 0,C 180,E1 -3691.479,E2 -3691.479} C_VEL
LIN {X 0,Y 544.65,Z 631.81,A -85,B 0,C 180,E1 -3692.959,E2 -3692.959} C_VEL
LIN {X 0,Y 544.684,Z 628.895,A -85,B 0,C 180,E1 -3694.07,E2 -3694.07} C_VEL
LIN {X 0,Y 544.654,Z 624.948,A -85,B 0,C 180,E1 -3695.182,E2 -3695.182} C_VEL
LIN {X 0,Y 544.73,Z 619.643,A -85,B 0,C 180,E1 -3696.34,E2 -3696.34} C_VEL
LIN {X 0,Y 544.836,Z 613.466,A -85,B 0,C 180,E1 -3697.411,E2 -3697.411} C_VEL
LIN {X 0,Y 545.007,Z 605.477,A -85,B 0,C 180,E1 -3698.528,E2 -3698.528} C_VEL
LIN {X 0,Y 545.152,Z 597.333,A -85,B 0,C 180,E1 -3699.461,E2 -3699.461} C_VEL
LIN {X 0,Y 545.361,Z 587.398,A -85,B 0,C 180,E1 -3700.394,E2 -3700.394} C_VEL
LIN {X 0,Y 545.553,Z 576.538,A -85,B 0,C 180,E1 -3701.212,E2 -3701.212} C_VEL
LIN {X 0,Y 545.767,Z 565.172,A -85,B 0,C 180,E1 -3701.89,E2 -3701.89} C_VEL
LIN {X 0,Y 545.949,Z 552.973,A -85,B 0,C 180,E1 -3702.452,E2 -3702.452} C_VEL
LIN {X 0,Y 546.099,Z 540.176,A -85,B 0,C 180,E1 -3702.874,E2 -3702.874} C_VEL
LIN {X 0,Y 546.258,Z 526.604,A -85,B 0,C 180,E1 -3703.153,E2 -3703.153} C_VEL
LIN {X 0,Y 546.495,Z 430.499,A -85,B 0,C 180,E1 -3704.425,E2 -3704.425} C_VEL
LIN {X 0,Y 545.358,Z 423.298,A -85,B 0,C 180,E1 -3704.577,E2 -3704.577} C_VEL
LIN {X 0,Y 545.648,Z 403.019,A -85,B 0,C 180,E1 -3707.741,E2 -3707.741} C_VEL
LIN {X 0,Y 546.002,Z 384.397,A -85,B 0,C 180,E1 -3710.73,E2 -3710.73} C_VEL
LIN {X 0,Y 546.025,Z 376.201,A -85,B 0,C 180,E1 -3712.069,E2 -3712.069} C_VEL
LIN {X 0,Y 545.097,Z 371.163,A -85,B 0,C 180,E1 -3712.98,E2 -3712.98} C_VEL
LIN {X 0,Y 545.082,Z 371.086,A -85,B 0,C 180,E1 -3716,E2 -3716} C_VEL
LIN {X 0,Y 545.091,Z 371.083,A -85,B 0,C 180,E1 -3718.748,E2 -3718.748} C_VEL
LIN {X 0,Y 545.079,Z 371.088,A -85,B 0,C 180,E1 -3721.682,E2 -3721.682} C_VEL
LIN {X 0,Y 545.083,Z 371.082,A -85,B 0,C 180,E1 -3724.562,E2 -3724.562} C_VEL
LIN {X 0,Y 545.068,Z 371.092,A -85,B 0,C 180,E1 -3727.301,E2 -3727.301} C_VEL
LIN {X 0,Y 545.074,Z 371.084,A -85,B 0,C 180,E1 -3730.141,E2 -3730.141} C_VEL
LIN {X 0,Y 545.085,Z 371.089,A -85,B 0,C 180,E1 -3733.105,E2 -3733.105} C_VEL
LIN {X 0,Y 545.064,Z 371.085,A -85,B 0,C 180,E1 -3736.224,E2 -3736.224} C_VEL
LIN {X 0,Y 545.121,Z 371.083,A -85,B 0,C 180,E1 -3738.889,E2 -3738.889} C_VEL
LIN {X 0,Y 545.052,Z 371.088,A -85,B 0,C 180,E1 -3741.762,E2 -3741.762} C_VEL
LIN {X 0,Y 545.061,Z 371.088,A -85,B 0,C 180,E1 -3744.533,E2 -3744.533} C_VEL
LIN {X 0,Y 545.078,Z 371.089,A -85,B 0,C 180,E1 -3747.212,E2 -3747.212} C_VEL
LIN {X 0,Y 545.062,Z 371.086,A -85,B 0,C 180,E1 -3749.81,E2 -3749.81} C_VEL
LIN {X 0,Y 545.091,Z 371.084,A -85,B 0,C 180,E1 -3752.344,E2 -3752.344} C_VEL
LIN {X 0,Y 545.113,Z 371.086,A -85,B 0,C 180,E1 -3754.82,E2 -3754.82} C_VEL
LIN {X 0,Y 545.039,Z 371.092,A -85,B 0,C 180,E1 -3757.242,E2 -3757.242} C_VEL
LIN {X 0,Y 545.115,Z 371.084,A -85,B 0,C 180,E1 -3760.415,E2 -3760.415} C_VEL
LIN {X 0,Y 545.071,Z 371.085,A -85,B 0,C 180,E1 -3763.521,E2 -3763.521} C_VEL
LIN {X 0,Y 545.089,Z 371.083,A -85,B 0,C 180,E1 -3765.82,E2 -3765.82} C_VEL
LIN {X 0,Y 545.111,Z 371.085,A -85,B 0,C 180,E1 -3768.849,E2 -3768.849} C_VEL
LIN {X 0,Y 545.124,Z 371.079,A -85,B 0,C 180,E1 -3771.847,E2 -3771.847} C_VEL
LIN {X 0,Y 545.201,Z 371.073,A -85,B 0,C 180,E1 -3774.823,E2 -3774.823} C_VEL
LIN {X 0,Y 545.188,Z 371.071,A -85,B 0,C 180,E1 -3777.784,E2 -3777.784} C_VEL
LIN {X 0,Y 545.209,Z 371.072,A -85,B 0,C 180,E1 -3780.739,E2 -3780.739} C_VEL
LIN {X 0,Y 545.17,Z 371.074,A -85,B 0,C 180,E1 -3782.956,E2 -3782.956} C_VEL
LIN {X 0,Y 545.166,Z 371.077,A -85,B 0,C 180,E1 -3785.919,E2 -3785.919} C_VEL
LIN {X 0,Y 545.115,Z 371.08,A -85,B 0,C 180,E1 -3788.9,E2 -3788.9} C_VEL
LIN {X 0,Y 545.128,Z 371.083,A -85,B 0,C 180,E1 -3791.904,E2 -3791.904} C_VEL
LIN {X 0,Y 545.08,Z 371.084,A -85,B 0,C 180,E1 -3794.944,E2 -3794.944} C_VEL
LIN {X 0,Y 545.078,Z 371.091,A -85,B 0,C 180,E1 -3798.026,E2 -3798.026} C_VEL
LIN {X 0,Y 545.093,Z 371.086,A -85,B 0,C 180,E1 -3800.372,E2 -3800.372} C_VEL
LIN {X 0,Y 545.086,Z 371.086,A -85,B 0,C 180,E1 -3803.559,E2 -3803.559} C_VEL
LIN {X 0,Y 545.084,Z 371.089,A -85,B 0,C 180,E1 -3806,E2 -3806} C_VEL
LIN {X 0,Y 545.088,Z 371.083,A -85,B 0,C 180,E1 -3808.749,E2 -3808.749} C_VEL
LIN {X 0,Y 545.074,Z 371.092,A -85,B 0,C 180,E1 -3811.683,E2 -3811.683} C_VEL
LIN {X 0,Y 545.08,Z 371.084,A -85,B 0,C 180,E1 -3814.563,E2 -3814.563} C_VEL
LIN {X 0,Y 545.061,Z 371.087,A -85,B 0,C 180,E1 -3817.017,E2 -3817.017} C_VEL
LIN {X 0,Y 544.354,Z 371.181,A -85,B 0,C 180,E1 -3817.634,E2 -3817.634} C_VEL
LIN {X 0,Y 541.491,Z 371.537,A -85,B 0,C 180,E1 -3818.635,E2 -3818.635} C_VEL
LIN {X 0,Y 539.105,Z 371.834,A -85,B 0,C 180,E1 -3819.441,E2 -3819.441} C_VEL
LIN {X 0,Y 538.095,Z 371.957,A -85,B 0,C 180,E1 -3820.063,E2 -3820.063} C_VEL
LIN {X 0,Y 538.019,Z 371.964,A -85,B 0,C 180,E1 -3820.273,E2 -3820.273} C_VEL
LIN {X 0,Y 538.03,Z 371.963,A -85,B 0,C 180,E1 -3822.989,E2 -3822.989} C_VEL
LIN {X 0,Y 538.027,Z 371.966,A -85,B 0,C 180,E1 -3825.926,E2 -3825.926} C_VEL
LIN {X 0,Y 538.077,Z 371.961,A -85,B 0,C 180,E1 -3829.249,E2 -3829.249} C_VEL
LIN {X 0,Y 537.993,Z 371.967,A -85,B 0,C 180,E1 -3832.123,E2 -3832.123} C_VEL
LIN {X 0,Y 538.02,Z 371.965,A -85,B 0,C 180,E1 -3834.918,E2 -3834.918} C_VEL
LIN {X 0,Y 538.026,Z 371.967,A -85,B 0,C 180,E1 -3837.618,E2 -3837.618} C_VEL
LIN {X 0,Y 538.018,Z 371.963,A -85,B 0,C 180,E1 -3840.239,E2 -3840.239} C_VEL
LIN {X 0,Y 538.058,Z 371.961,A -85,B 0,C 180,E1 -3842.796,E2 -3842.796} C_VEL
LIN {X 0,Y 538.049,Z 371.966,A -85,B 0,C 180,E1 -3845.293,E2 -3845.293} C_VEL
LIN {X 0,Y 538.023,Z 371.963,A -85,B 0,C 180,E1 -3848.546,E2 -3848.546} C_VEL
LIN {X 0,Y 538.035,Z 371.967,A -85,B 0,C 180,E1 -3850.94,E2 -3850.94} C_VEL
LIN {X 0,Y 538.025,Z 371.967,A -85,B 0,C 180,E1 -3853.299,E2 -3853.299} C_VEL
LIN {X 0,Y 538.066,Z 371.958,A -85,B 0,C 180,E1 -3855.631,E2 -3855.631} C_VEL
LIN {X 0,Y 538.08,Z 371.962,A -85,B 0,C 180,E1 -3858.702,E2 -3858.702} C_VEL
LIN {X 0,Y 538.099,Z 372.134,A -85,B 0,C 180,E1 -3861.669,E2 -3861.669} C_VEL
LIN {X 0,Y 538.842,Z 377.777,A -85,B 0,C 180,E1 -3862.739,E2 -3862.739} C_VEL
LIN {X 0,Y 538.549,Z 392.141,A -85,B 0,C 180,E1 -3865.322,E2 -3865.322} C_VEL
LIN {X 0,Y 538.321,Z 408.984,A -85,B 0,C 180,E1 -3868.27,E2 -3868.27} C_VEL
LIN {X 0,Y 538.72,Z 411.736,A -85,B 0,C 180,E1 -3868.354,E2 -3868.354} C_VEL
LIN {X 0,Y 539.687,Z 417.614,A -85,B 0,C 180,E1 -3868.461,E2 -3868.461} C_VEL
LIN {X 0,Y 539.291,Z 515.974,A -85,B 0,C 180,E1 -3869.79,E2 -3869.79} C_VEL
LIN {X 0,Y 539.178,Z 529.061,A -85,B 0,C 180,E1 -3870.117,E2 -3870.117} C_VEL
LIN {X 0,Y 538.945,Z 542.238,A -85,B 0,C 180,E1 -3870.607,E2 -3870.607} C_VEL
LIN {X 0,Y 538.691,Z 554.122,A -85,B 0,C 180,E1 -3871.215,E2 -3871.215} C_VEL
LIN {X 0,Y 538.446,Z 565.475,A -85,B 0,C 180,E1 -3871.963,E2 -3871.963} C_VEL
LIN {X 0,Y 538.199,Z 575.739,A -85,B 0,C 180,E1 -3872.807,E2 -3872.807} C_VEL
LIN {X 0,Y 537.983,Z 585.005,A -85,B 0,C 180,E1 -3873.745,E2 -3873.745} C_VEL
LIN {X 0,Y 537.849,Z 593.985,A -85,B 0,C 180,E1 -3874.872,E2 -3874.872} C_VEL
LIN {X 0,Y 537.729,Z 601.263,A -85,B 0,C 180,E1 -3876.001,E2 -3876.001} C_VEL
LIN {X 0,Y 537.642,Z 607.115,A -85,B 0,C 180,E1 -3877.133,E2 -3877.133} C_VEL
LIN {X 0,Y 537.601,Z 611.738,A -85,B 0,C 180,E1 -3878.268,E2 -3878.268} C_VEL
LIN {X 0,Y 537.53,Z 615.269,A -85,B 0,C 180,E1 -3879.406,E2 -3879.406} C_VEL
LIN {X 0,Y 537.493,Z 617.784,A -85,B 0,C 180,E1 -3880.547,E2 -3880.547} C_VEL
LIN {X 0,Y 537.538,Z 618.93,A -85,B 0,C 180,E1 -3881.31,E2 -3881.31} C_VEL
LIN {X 0,Y 537.473,Z 619.964,A -85,B 0,C 180,E1 -3882.843,E2 -3882.843} C_VEL
LIN {X 0,Y 537.475,Z 619.884,A -85,B 0,C 180,E1 -3883.613,E2 -3883.613} C_VEL
LIN {X 0,Y 537.483,Z 619.097,A -85,B 0,C 180,E1 -3884.623,E2 -3884.623} C_VEL
LIN {X 0,Y 537.458,Z 617.016,A -85,B 0,C 180,E1 -3885.938,E2 -3885.938} C_VEL
LIN {X 0,Y 537.523,Z 615.175,A -85,B 0,C 180,E1 -3886.716,E2 -3886.716} C_VEL
LIN {X 0,Y 537.589,Z 611.481,A -85,B 0,C 180,E1 -3887.891,E2 -3887.891} C_VEL
LIN {X 0,Y 537.651,Z 606.555,A -85,B 0,C 180,E1 -3889.074,E2 -3889.074} C_VEL
LIN {X 0,Y 537.741,Z 600.229,A -85,B 0,C 180,E1 -3890.263,E2 -3890.263} C_VEL
LIN {X 0,Y 537.9,Z 592.255,A -85,B 0,C 180,E1 -3891.458,E2 -3891.458} C_VEL
LIN {X 0,Y 538.077,Z 583.949,A -85,B 0,C 180,E1 -3892.46,E2 -3892.46} C_VEL
LIN {X 0,Y 538.294,Z 573.674,A -85,B 0,C 180,E1 -3893.466,E2 -3893.466} C_VEL
LIN {X 0,Y 538.507,Z 563.903,A -85,B 0,C 180,E1 -3894.242,E2 -3894.242} C_VEL
LIN {X 0,Y 538.739,Z 552.269,A -85,B 0,C 180,E1 -3894.982,E2 -3894.982} C_VEL
LIN {X 0,Y 538.969,Z 540.723,A -85,B 0,C 180,E1 -3895.547,E2 -3895.547} C_VEL
LIN {X 0,Y 539.207,Z 527.31,A -85,B 0,C 180,E1 -3896.028,E2 -3896.028} C_VEL
LIN {X 0,Y 539.324,Z 514.558,A -85,B 0,C 180,E1 -3896.324,E2 -3896.324} C_VEL
LIN {X 0,Y 539.668,Z 417.657,A -85,B 0,C 180,E1 -3897.629,E2 -3897.629} C_VEL
LIN {X 0,Y 538.266,Z 409.21,A -85,B 0,C 180,E1 -3897.806,E2 -3897.806} C_VEL
LIN {X 0,Y 538.271,Z 406.394,A -85,B 0,C 180,E1 -3898.248,E2 -3898.248} C_VEL
LIN {X 0,Y 538.553,Z 390.737,A -85,B 0,C 180,E1 -3901.028,E2 -3901.028} C_VEL
LIN {X 0,Y 538.872,Z 377.421,A -85,B 0,C 180,E1 -3903.416,E2 -3903.416} C_VEL
LIN {X 0,Y 538.064,Z 372.006,A -85,B 0,C 180,E1 -3904.476,E2 -3904.476} C_VEL
LIN {X 0,Y 538.023,Z 371.97,A -85,B 0,C 180,E1 -3907.172,E2 -3907.172} C_VEL
LIN {X 0,Y 538.051,Z 371.961,A -85,B 0,C 180,E1 -3909.793,E2 -3909.793} C_VEL
LIN {X 0,Y 538.019,Z 371.967,A -85,B 0,C 180,E1 -3912.785,E2 -3912.785} C_VEL
LIN {X 0,Y 538.025,Z 371.962,A -85,B 0,C 180,E1 -3915.924,E2 -3915.924} C_VEL
LIN {X 0,Y 538.075,Z 371.963,A -85,B 0,C 180,E1 -3919.248,E2 -3919.248} C_VEL
LIN {X 0,Y 537.996,Z 371.964,A -85,B 0,C 180,E1 -3922.123,E2 -3922.123} C_VEL
LIN {X 0,Y 538.015,Z 371.969,A -85,B 0,C 180,E1 -3924.917,E2 -3924.917} C_VEL
LIN {X 0,Y 538.025,Z 371.963,A -85,B 0,C 180,E1 -3927.618,E2 -3927.618} C_VEL
LIN {X 0,Y 538.036,Z 371.956,A -85,B 0,C 180,E1 -3930.24,E2 -3930.24} C_VEL
LIN {X 0,Y 538.064,Z 371.962,A -85,B 0,C 180,E1 -3932.796,E2 -3932.796} C_VEL
LIN {X 0,Y 538.045,Z 371.964,A -85,B 0,C 180,E1 -3935.292,E2 -3935.292} C_VEL
LIN {X 0,Y 538.023,Z 371.96,A -85,B 0,C 180,E1 -3938.037,E2 -3938.037} C_VEL
LIN {X 0,Y 538.037,Z 371.967,A -85,B 0,C 180,E1 -3940.94,E2 -3940.94} C_VEL
LIN {X 0,Y 538.021,Z 371.966,A -85,B 0,C 180,E1 -3943.299,E2 -3943.299} C_VEL
LIN {X 0,Y 538.055,Z 371.957,A -85,B 0,C 180,E1 -3945.63,E2 -3945.63} C_VEL
LIN {X 0,Y 538.081,Z 371.961,A -85,B 0,C 180,E1 -3948.702,E2 -3948.702} C_VEL
LIN {X 0,Y 538.084,Z 371.954,A -85,B 0,C 180,E1 -3951.74,E2 -3951.74} C_VEL
LIN {X 0,Y 538.177,Z 371.948,A -85,B 0,C 180,E1 -3954.755,E2 -3954.755} C_VEL
LIN {X 0,Y 538.159,Z 371.944,A -85,B 0,C 180,E1 -3957.755,E2 -3957.755} C_VEL
LIN {X 0,Y 538.18,Z 371.949,A -85,B 0,C 180,E1 -3960.748,E2 -3960.748} C_VEL
LIN {X 0,Y 538.137,Z 371.951,A -85,B 0,C 180,E1 -3962.995,E2 -3962.995} C_VEL
LIN {X 0,Y 538.116,Z 371.95,A -85,B 0,C 180,E1 -3965.997,E2 -3965.997} C_VEL
LIN {X 0,Y 538.07,Z 371.96,A -85,B 0,C 180,E1 -3969.018,E2 -3969.018} C_VEL
LIN {X 0,Y 538.075,Z 371.956,A -85,B 0,C 180,E1 -3972.063,E2 -3972.063} C_VEL
LIN {X 0,Y 538.037,Z 371.963,A -85,B 0,C 180,E1 -3975.144,E2 -3975.144} C_VEL
LIN {X 0,Y 538.028,Z 371.962,A -85,B 0,C 180,E1 -3978.27,E2 -3978.27} C_VEL
LIN {X 0,Y 538.035,Z 371.969,A -85,B 0,C 180,E1 -3980.652,E2 -3980.652} C_VEL
LIN {X 0,Y 538.033,Z 371.96,A -85,B 0,C 180,E1 -3983.887,E2 -3983.887} C_VEL
LIN {X 0,Y 538.043,Z 371.963,A -85,B 0,C 180,E1 -3986.367,E2 -3986.367} C_VEL
LIN {X 0,Y 538.025,Z 371.966,A -85,B 0,C 180,E1 -3988.935,E2 -3988.935} C_VEL
LIN {X 0,Y 538.021,Z 371.962,A -85,B 0,C 180,E1 -3991.891,E2 -3991.891} C_VEL
LIN {X 0,Y 538.028,Z 371.969,A -85,B 0,C 180,E1 -3994.622,E2 -3994.622} C_VEL
LIN {X 0,Y 538.005,Z 371.964,A -85,B 0,C 180,E1 -3997.172,E2 -3997.172} C_VEL
LIN {X 0,Y 538.05,Z 371.958,A -85,B 0,C 180,E1 -3999.795,E2 -3999.795} C_VEL
LIN {X 0,Y 538.021,Z 371.968,A -85,B 0,C 180,E1 -4002.786,E2 -4002.786} C_VEL
LIN {X 0,Y 538.025,Z 371.961,A -85,B 0,C 180,E1 -4005.926,E2 -4005.926} C_VEL
LIN {X 0,Y 538.049,Z 371.958,A -85,B 0,C 180,E1 -4009.225,E2 -4009.225} C_VEL
LIN {X 0,Y 537.992,Z 371.97,A -85,B 0,C 180,E1 -4012.123,E2 -4012.123} C_VEL
LIN {X 0,Y 538.021,Z 371.965,A -85,B 0,C 180,E1 -4014.918,E2 -4014.918} C_VEL
LIN {X 0,Y 538.031,Z 371.962,A -85,B 0,C 180,E1 -4017.619,E2 -4017.619} C_VEL
LIN {X 0,Y 538.018,Z 371.97,A -85,B 0,C 180,E1 -4020.24,E2 -4020.24} C_VEL
LIN {X 0,Y 538.07,Z 371.961,A -85,B 0,C 180,E1 -4022.797,E2 -4022.797} C_VEL
LIN {X 0,Y 538.051,Z 371.963,A -85,B 0,C 180,E1 -4025.293,E2 -4025.293} C_VEL
LIN {X 0,Y 538.076,Z 372.066,A -85,B 0,C 180,E1 -4026.881,E2 -4026.881} C_VEL
LIN {X 0,Y 539.079,Z 377.776,A -85,B 0,C 180,E1 -4027.909,E2 -4027.909} C_VEL
LIN {X 0,Y 538.88,Z 391.568,A -85,B 0,C 180,E1 -4030.179,E2 -4030.179} C_VEL
LIN {X 0,Y 538.522,Z 408.558,A -85,B 0,C 180,E1 -4032.925,E2 -4032.925} C_VEL
LIN {X 0,Y 538.36,Z 423.224,A -85,B 0,C 180,E1 -4035.232,E2 -4035.232} C_VEL
LIN {X 0,Y 539.671,Z 432.2,A -85,B 0,C 180,E1 -4035.413,E2 -4035.413} C_VEL
LIN {X 0,Y 539.34,Z 530.869,A -85,B 0,C 180,E1 -4036.747,E2 -4036.747} C_VEL
LIN {X 0,Y 539.181,Z 544.15,A -85,B 0,C 180,E1 -4037.078,E2 -4037.078} C_VEL
LIN {X 0,Y 538.947,Z 557.436,A -85,B 0,C 180,E1 -4037.575,E2 -4037.575} C_VEL
LIN {X 0,Y 538.741,Z 569.326,A -85,B 0,C 180,E1 -4038.189,E2 -4038.189} C_VEL
LIN {X 0,Y 538.5,Z 581.467,A -85,B 0,C 180,E1 -4038.997,E2 -4038.997} C_VEL
LIN {X 0,Y 538.228,Z 591.647,A -85,B 0,C 180,E1 -4039.847,E2 -4039.847} C_VEL
LIN {X 0,Y 538.026,Z 600.789,A -85,B 0,C 180,E1 -4040.793,E2 -4040.793} C_VEL
LIN {X 0,Y 537.85,Z 609.69,A -85,B 0,C 180,E1 -4041.925,E2 -4041.925} C_VEL
LIN {X 0,Y 537.728,Z 616.85,A -85,B 0,C 180,E1 -4043.057,E2 -4043.057} C_VEL
LIN {X 0,Y 537.676,Z 623.367,A -85,B 0,C 180,E1 -4044.374,E2 -4044.374} C_VEL
LIN {X 0,Y 537.557,Z 627.677,A -85,B 0,C 180,E1 -4045.501,E2 -4045.501} C_VEL
LIN {X 0,Y 537.591,Z 629.958,A -85,B 0,C 180,E1 -4046.252,E2 -4046.252} C_VEL
LIN {X 0,Y 537.551,Z 631.807,A -85,B 0,C 180,E1 -4047.003,E2 -4047.003} C_VEL
LIN {X 0,Y 537.451,Z 634.182,A -85,B 0,C 180,E1 -4048.502,E2 -4048.502} C_VEL
LIN {X 0,Y 537.442,Z 635,A -85,B 0,C 180,E1 -4050,E2 -4050} C_VEL
LIN {X 0,Y 537.451,Z 634.183,A -85,B 0,C 180,E1 -4051.499,E2 -4051.499} C_VEL
LIN {X 0,Y 537.551,Z 631.81,A -85,B 0,C 180,E1 -4052.998,E2 -4052.998} C_VEL
LIN {X 0,Y 537.603,Z 628.895,A -85,B 0,C 180,E1 -4054.123,E2 -4054.123} C_VEL
LIN {X 0,Y 537.588,Z 624.948,A -85,B 0,C 180,E1 -4055.251,E2 -4055.251} C_VEL
LIN {X 0,Y 537.645,Z 620.125,A -85,B 0,C 180,E1 -4056.326,E2 -4056.326} C_VEL
LIN {X 0,Y 537.791,Z 613.466,A -85,B 0,C 180,E1 -4057.509,E2 -4057.509} C_VEL
LIN {X 0,Y 537.972,Z 605.477,A -85,B 0,C 180,E1 -4058.641,E2 -4058.641} C_VEL
LIN {X 0,Y 538.143,Z 597.333,A -85,B 0,C 180,E1 -4059.585,E2 -4059.585} C_VEL
LIN {X 0,Y 538.35,Z 587.386,A -85,B 0,C 180,E1 -4060.531,E2 -4060.531} C_VEL
LIN {X 0,Y 538.566,Z 577.564,A -85,B 0,C 180,E1 -4061.288,E2 -4061.288} C_VEL
LIN {X 0,Y 538.774,Z 566.955,A -85,B 0,C 180,E1 -4061.948,E2 -4061.948} C_VEL
LIN {X 0,Y 538.977,Z 554.037,A -85,B 0,C 180,E1 -4062.568,E2 -4062.568} C_VEL
LIN {X 0,Y 539.175,Z 541.005,A -85,B 0,C 180,E1 -4063.018,E2 -4063.018} C_VEL
LIN {X 0,Y 539.353,Z 528.004,A -85,B 0,C 180,E1 -4063.301,E2 -4063.301} C_VEL
LIN {X 0,Y 539.559,Z 430.86,A -85,B 0,C 180,E1 -4064.608,E2 -4064.608} C_VEL
LIN {X 0,Y 538.368,Z 423.294,A -85,B 0,C 180,E1 -4064.764,E2 -4064.764} C_VEL
LIN {X 0,Y 538.359,Z 418.248,A -85,B 0,C 180,E1 -4065.522,E2 -4065.522} C_VEL
LIN {X 0,Y 538.709,Z 400.072,A -85,B 0,C 180,E1 -4068.443,E2 -4068.443} C_VEL
LIN {X 0,Y 539.1,Z 381.901,A -85,B 0,C 180,E1 -4071.409,E2 -4071.409} C_VEL
LIN {X 0,Y 539.008,Z 377.058,A -85,B 0,C 180,E1 -4072.217,E2 -4072.217} C_VEL
LIN {X 0,Y 538.071,Z 372.035,A -85,B 0,C 180,E1 -4073.145,E2 -4073.145} C_VEL
LIN {X 0,Y 538.046,Z 371.967,A -85,B 0,C 180,E1 -4075.672,E2 -4075.672} C_VEL
LIN {X 0,Y 538.046,Z 371.962,A -85,B 0,C 180,E1 -4078.049,E2 -4078.049} C_VEL
LIN {X 0,Y 538.022,Z 371.962,A -85,B 0,C 180,E1 -4080.626,E2 -4080.626} C_VEL
LIN {X 0,Y 538.045,Z 371.966,A -85,B 0,C 180,E1 -4083.282,E2 -4083.282} C_VEL
LIN {X 0,Y 538.028,Z 371.962,A -85,B 0,C 180,E1 -4086.001,E2 -4086.001} C_VEL
LIN {X 0,Y 538.015,Z 371.965,A -85,B 0,C 180,E1 -4088.83,E2 -4088.83} C_VEL
LIN {X 0,Y 538.037,Z 371.962,A -85,B 0,C 180,E1 -4091.879,E2 -4091.879} C_VEL
LIN {X 0,Y 538.031,Z 371.968,A -85,B 0,C 180,E1 -4095.14,E2 -4095.14} C_VEL
LIN {X 0,Y 538.057,Z 371.958,A -85,B 0,C 180,E1 -4098.229,E2 -4098.229} C_VEL
LIN {X 0,Y 538.013,Z 371.972,A -85,B 0,C 180,E1 -4101.169,E2 -4101.169} C_VEL
LIN {X 0,Y 538.026,Z 371.962,A -85,B 0,C 180,E1 -4104.083,E2 -4104.083} C_VEL
LIN {X 0,Y 538.028,Z 371.967,A -85,B 0,C 180,E1 -4106.727,E2 -4106.727} C_VEL
LIN {X 0,Y 538.021,Z 371.964,A -85,B 0,C 180,E1 -4109.556,E2 -4109.556} C_VEL
LIN {X 0,Y 538.043,Z 371.96,A -85,B 0,C 180,E1 -4111.95,E2 -4111.95} C_VEL
LIN {X 0,Y 538.071,Z 371.961,A -85,B 0,C 180,E1 -4114.467,E2 -4114.467} C_VEL
LIN {X 0,Y 538.017,Z 371.971,A -85,B 0,C 180,E1 -4116.928,E2 -4116.928} C_VEL
LIN {X 0,Y 538.073,Z 371.958,A -85,B 0,C 180,E1 -4120.148,E2 -4120.148} C_VEL
LIN {X 0,Y 538.022,Z 371.964,A -85,B 0,C 180,E1 -4123.299,E2 -4123.299} C_VEL
LIN {X 0,Y 538.058,Z 371.959,A -85,B 0,C 180,E1 -4125.63,E2 -4125.63} C_VEL
LIN {X 0,Y 538.071,Z 371.964,A -85,B 0,C 180,E1 -4128.701,E2 -4128.701} C_VEL
LIN {X 0,Y 538.081,Z 371.956,A -85,B 0,C 180,E1 -4131.739,E2 -4131.739} C_VEL
LIN {X 0,Y 538.158,Z 371.951,A -85,B 0,C 180,E1 -4134.755,E2 -4134.755} C_VEL
LIN {X 0,Y 538.16,Z 371.947,A -85,B 0,C 180,E1 -4137.755,E2 -4137.755} C_VEL
LIN {X 0,Y 538.179,Z 371.947,A -85,B 0,C 180,E1 -4140.748,E2 -4140.748} C_VEL
LIN {X 0,Y 538.136,Z 371.95,A -85,B 0,C 180,E1 -4142.994,E2 -4142.994} C_VEL
LIN {X 0,Y 538.118,Z 371.956,A -85,B 0,C 180,E1 -4145.997,E2 -4145.997} C_VEL
LIN {X 0,Y 538.066,Z 371.958,A -85,B 0,C 180,E1 -4149.018,E2 -4149.018} C_VEL
LIN {X 0,Y 538.077,Z 371.962,A -85,B 0,C 180,E1 -4152.063,E2 -4152.063} C_VEL
LIN {X 0,Y 538.04,Z 371.961,A -85,B 0,C 180,E1 -4155.144,E2 -4155.144} C_VEL
LIN {X 0,Y 538.03,Z 371.968,A -85,B 0,C 180,E1 -4158.27,E2 -4158.27} C_VEL
LIN {X 0,Y 538.037,Z 371.962,A -85,B 0,C 180,E1 -4160.651,E2 -4160.651} C_VEL
LIN {X 0,Y 538.018,Z 371.97,A -85,B 0,C 180,E1 -4163.888,E2 -4163.888} C_VEL
LIN {X 0,Y 538.045,Z 371.963,A -85,B 0,C 180,E1 -4166.367,E2 -4166.367} C_VEL
LIN {X 0,Y 538.051,Z 371.959,A -85,B 0,C 180,E1 -4168.939,E2 -4168.939} C_VEL
LIN {X 0,Y 538.024,Z 371.969,A -85,B 0,C 180,E1 -4171.891,E2 -4171.891} C_VEL
LIN {X 0,Y 538.03,Z 371.962,A -85,B 0,C 180,E1 -4174.622,E2 -4174.622} C_VEL
LIN {X 0,Y 538.004,Z 371.967,A -85,B 0,C 180,E1 -4177.171,E2 -4177.171} C_VEL
LIN {X 0,Y 538.019,Z 371.964,A -85,B 0,C 180,E1 -4180.273,E2 -4180.273} C_VEL
LIN {X 0,Y 537.369,Z 372.045,A -85,B 0,C 180,E1 -4180.898,E2 -4180.898} C_VEL
LIN {X 0,Y 534.52,Z 372.407,A -85,B 0,C 180,E1 -4181.913,E2 -4181.913} C_VEL
LIN {X 0,Y 532.096,Z 372.713,A -85,B 0,C 180,E1 -4182.73,E2 -4182.73} C_VEL
LIN {X 0,Y 531.049,Z 372.841,A -85,B 0,C 180,E1 -4183.362,E2 -4183.362} C_VEL
LIN {X 0,Y 530.961,Z 372.849,A -85,B 0,C 180,E1 -4183.575,E2 -4183.575} C_VEL
LIN {X 0,Y 530.962,Z 372.842,A -85,B 0,C 180,E1 -4186.506,E2 -4186.506} C_VEL
LIN {X 0,Y 531.025,Z 372.84,A -85,B 0,C 180,E1 -4189.572,E2 -4189.572} C_VEL
LIN {X 0,Y 530.968,Z 372.841,A -85,B 0,C 180,E1 -4192.577,E2 -4192.577} C_VEL
LIN {X 0,Y 531.002,Z 372.845,A -85,B 0,C 180,E1 -4195.312,E2 -4195.312} C_VEL
LIN {X 0,Y 530.971,Z 372.842,A -85,B 0,C 180,E1 -4198.033,E2 -4198.033} C_VEL
LIN {X 0,Y 530.989,Z 372.842,A -85,B 0,C 180,E1 -4200.874,E2 -4200.874} C_VEL
LIN {X 0,Y 531.002,Z 372.844,A -85,B 0,C 180,E1 -4203.257,E2 -4203.257} C_VEL
LIN {X 0,Y 530.986,Z 372.839,A -85,B 0,C 180,E1 -4205.961,E2 -4205.961} C_VEL
LIN {X 0,Y 531,Z 372.845,A -85,B 0,C 180,E1 -4209.062,E2 -4209.062} C_VEL
LIN {X 0,Y 530.989,Z 372.841,A -85,B 0,C 180,E1 -4211.479,E2 -4211.479} C_VEL
LIN {X 0,Y 530.997,Z 372.84,A -85,B 0,C 180,E1 -4214.65,E2 -4214.65} C_VEL
LIN {X 0,Y 531.043,Z 372.834,A -85,B 0,C 180,E1 -4217.775,E2 -4217.775} C_VEL
LIN {X 0,Y 531.031,Z 372.841,A -85,B 0,C 180,E1 -4220.862,E2 -4220.862} C_VEL
LIN {X 0,Y 531.087,Z 373.06,A -85,B 0,C 180,E1 -4221.534,E2 -4221.534} C_VEL
LIN {X 0,Y 531.867,Z 378.826,A -85,B 0,C 180,E1 -4222.64,E2 -4222.64} C_VEL
LIN {X 0,Y 531.559,Z 393.206,A -85,B 0,C 180,E1 -4225.26,E2 -4225.26} C_VEL
LIN {X 0,Y 531.343,Z 409.197,A -85,B 0,C 180,E1 -4228.081,E2 -4228.081} C_VEL
LIN {X 0,Y 532.268,Z 414.815,A -85,B 0,C 180,E1 -4228.213,E2 -4228.213} C_VEL
LIN {X 0,Y 532.845,Z 419.887,A -85,B 0,C 180,E1 -4228.299,E2 -4228.299} C_VEL
LIN {X 0,Y 532.378,Z 516.372,A -85,B 0,C 180,E1 -4229.622,E2 -4229.622} C_VEL
LIN {X 0,Y 532.239,Z 530.112,A -85,B 0,C 180,E1 -4229.976,E2 -4229.976} C_VEL
LIN {X 0,Y 532.001,Z 543.006,A -85,B 0,C 180,E1 -4230.473,E2 -4230.473} C_VEL
LIN {X 0,Y 531.721,Z 555.49,A -85,B 0,C 180,E1 -4231.136,E2 -4231.136} C_VEL
LIN {X 0,Y 531.439,Z 566.619,A -85,B 0,C 180,E1 -4231.894,E2 -4231.894} C_VEL
LIN {X 0,Y 531.175,Z 576.684,A -85,B 0,C 180,E1 -4232.749,E2 -4232.749} C_VEL
LIN {X 0,Y 530.913,Z 586.575,A -85,B 0,C 180,E1 -4233.795,E2 -4233.795} C_VEL
LIN {X 0,Y 530.766,Z 595.298,A -85,B 0,C 180,E1 -4234.937,E2 -4234.937} C_VEL
LIN {X 0,Y 530.621,Z 602.315,A -85,B 0,C 180,E1 -4236.082,E2 -4236.082} C_VEL
LIN {X 0,Y 530.558,Z 607.928,A -85,B 0,C 180,E1 -4237.229,E2 -4237.229} C_VEL
LIN {X 0,Y 530.503,Z 612.363,A -85,B 0,C 180,E1 -4238.379,E2 -4238.379} C_VEL
LIN {X 0,Y 530.434,Z 614.714,A -85,B 0,C 180,E1 -4239.148,E2 -4239.148} C_VEL
LIN {X 0,Y 530.404,Z 616.634,A -85,B 0,C 180,E1 -4239.918,E2 -4239.918} C_VEL
LIN {X 0,Y 530.447,Z 619.013,A -85,B 0,C 180,E1 -4241.35,E2 -4241.35} C_VEL
LIN {X 0,Y 530.38,Z 619.77,A -85,B 0,C 180,E1 -4242.24,E2 -4242.24} C_VEL
LIN {X 0,Y 530.366,Z 620.012,A -85,B 0,C 180,E1 -4243.018,E2 -4243.018} C_VEL
LIN {X 0,Y 530.403,Z 619.802,A -85,B 0,C 180,E1 -4243.798,E2 -4243.798} C_VEL
LIN {X 0,Y 530.402,Z 619.055,A -85,B 0,C 180,E1 -4244.698,E2 -4244.698} C_VEL
LIN {X 0,Y 530.368,Z 616.666,A -85,B 0,C 180,E1 -4246.157,E2 -4246.157} C_VEL
LIN {X 0,Y 530.479,Z 613.155,A -85,B 0,C 180,E1 -4247.468,E2 -4247.468} C_VEL
LIN {X 0,Y 530.531,Z 609.297,A -85,B 0,C 180,E1 -4248.537,E2 -4248.537} C_VEL
LIN {X 0,Y 530.627,Z 602.96,A -85,B 0,C 180,E1 -4249.885,E2 -4249.885} C_VEL
LIN {X 0,Y 530.728,Z 596.652,A -85,B 0,C 180,E1 -4250.948,E2 -4250.948} C_VEL
LIN {X 0,Y 530.966,Z 588.233,A -85,B 0,C 180,E1 -4252.098,E2 -4252.098} C_VEL
LIN {X 0,Y 531.189,Z 578.329,A -85,B 0,C 180,E1 -4253.179,E2 -4253.179} C_VEL
LIN {X 0,Y 531.397,Z 569.145,A -85,B 0,C 180,E1 -4253.996,E2 -4253.996} C_VEL
LIN {X 0,Y 531.691,Z 557.797,A -85,B 0,C 180,E1 -4254.814,E2 -4254.814} C_VEL
LIN {X 0,Y 531.891,Z 545.825,A -85,B 0,C 180,E1 -4255.483,E2 -4255.483} C_VEL
LIN {X 0,Y 532.201,Z 533.473,A -85,B 0,C 180,E1 -4256.001,E2 -4256.001} C_VEL
LIN {X 0,Y 532.349,Z 520.82,A -85,B 0,C 180,E1 -4256.374,E2 -4256.374} C_VEL
LIN {X 0,Y 532.463,Z 504.969,A -85,B 0,C 180,E1 -4256.641,E2 -4256.641} C_VEL
LIN {X 0,Y 532.71,Z 417.713,A -85,B 0,C 180,E1 -4257.825,E2 -4257.825} C_VEL
LIN {X 0,Y 531.291,Z 409.479,A -85,B 0,C 180,E1 -4257.994,E2 -4257.994} C_VEL
LIN {X 0,Y 531.25,Z 408.191,A -85,B 0,C 180,E1 -4258.149,E2 -4258.149} C_VEL
LIN {X 0,Y 531.564,Z 392.103,A -85,B 0,C 180,E1 -4261.039,E2 -4261.039} C_VEL
LIN {X 0,Y 531.923,Z 378.862,A -85,B 0,C 180,E1 -4263.443,E2 -4263.443} C_VEL
LIN {X 0,Y 530.982,Z 372.886,A -85,B 0,C 180,E1 -4264.632,E2 -4264.632} C_VEL
LIN {X 0,Y 530.971,Z 372.846,A -85,B 0,C 180,E1 -4267.506,E2 -4267.506} C_VEL
LIN {X 0,Y 531.004,Z 372.839,A -85,B 0,C 180,E1 -4270.43,E2 -4270.43} C_VEL
LIN {X 0,Y 530.962,Z 372.846,A -85,B 0,C 180,E1 -4273.494,E2 -4273.494} C_VEL
LIN {X 0,Y 530.963,Z 372.843,A -85,B 0,C 180,E1 -4276.505,E2 -4276.505} C_VEL
LIN {X 0,Y 531.004,Z 372.839,A -85,B 0,C 180,E1 -4279.569,E2 -4279.569} C_VEL
LIN {X 0,Y 530.971,Z 372.842,A -85,B 0,C 180,E1 -4282.575,E2 -4282.575} C_VEL
LIN {X 0,Y 530.997,Z 372.84,A -85,B 0,C 180,E1 -4285.311,E2 -4285.311} C_VEL
LIN {X 0,Y 530.976,Z 372.84,A -85,B 0,C 180,E1 -4288.032,E2 -4288.032} C_VEL
LIN {X 0,Y 530.999,Z 372.838,A -85,B 0,C 180,E1 -4290.87,E2 -4290.87} C_VEL
LIN {X 0,Y 531.004,Z 372.841,A -85,B 0,C 180,E1 -4293.256,E2 -4293.256} C_VEL
LIN {X 0,Y 530.999,Z 372.837,A -85,B 0,C 180,E1 -4295.955,E2 -4295.955} C_VEL
LIN {X 0,Y 530.997,Z 372.845,A -85,B 0,C 180,E1 -4299.062,E2 -4299.062} C_VEL
LIN {X 0,Y 531.007,Z 372.835,A -85,B 0,C 180,E1 -4302.277,E2 -4302.277} C_VEL
LIN {X 0,Y 531.01,Z 372.836,A -85,B 0,C 180,E1 -4305.436,E2 -4305.436} C_VEL
LIN {X 0,Y 531.037,Z 372.836,A -85,B 0,C 180,E1 -4308.55,E2 -4308.55} C_VEL
LIN {X 0,Y 531.053,Z 372.83,A -85,B 0,C 180,E1 -4311.629,E2 -4311.629} C_VEL
LIN {X 0,Y 531.133,Z 372.824,A -85,B 0,C 180,E1 -4314.685,E2 -4314.685} C_VEL
LIN {X 0,Y 531.131,Z 372.819,A -85,B 0,C 180,E1 -4317.725,E2 -4317.725} C_VEL
LIN {X 0,Y 531.149,Z 372.825,A -85,B 0,C 180,E1 -4320.758,E2 -4320.758} C_VEL
LIN {X 0,Y 531.103,Z 372.826,A -85,B 0,C 180,E1 -4323.034,E2 -4323.034} C_VEL
LIN {X 0,Y 531.076,Z 372.827,A -85,B 0,C 180,E1 -4326.077,E2 -4326.077} C_VEL
LIN {X 0,Y 531.029,Z 372.835,A -85,B 0,C 180,E1 -4329.138,E2 -4329.138} C_VEL
LIN {X 0,Y 531.032,Z 372.834,A -85,B 0,C 180,E1 -4332.225,E2 -4332.225} C_VEL
LIN {X 0,Y 530.988,Z 372.839,A -85,B 0,C 180,E1 -4335.35,E2 -4335.35} C_VEL
LIN {X 0,Y 531.008,Z 372.834,A -85,B 0,C 180,E1 -4337.723,E2 -4337.723} C_VEL
LIN {X 0,Y 530.997,Z 372.841,A -85,B 0,C 180,E1 -4340.938,E2 -4340.938} C_VEL
LIN {X 0,Y 530.999,Z 372.837,A -85,B 0,C 180,E1 -4344.046,E2 -4344.046} C_VEL
LIN {X 0,Y 531.005,Z 372.842,A -85,B 0,C 180,E1 -4346.744,E2 -4346.744} C_VEL
LIN {X 0,Y 530.976,Z 372.84,A -85,B 0,C 180,E1 -4349.323,E2 -4349.323} C_VEL
LIN {X 0,Y 530.974,Z 372.842,A -85,B 0,C 180,E1 -4352.104,E2 -4352.104} C_VEL
LIN {X 0,Y 530.985,Z 372.844,A -85,B 0,C 180,E1 -4354.855,E2 -4354.855} C_VEL
LIN {X 0,Y 530.962,Z 372.84,A -85,B 0,C 180,E1 -4357.508,E2 -4357.508} C_VEL
LIN {X 0,Y 531.022,Z 372.841,A -85,B 0,C 180,E1 -4360.429,E2 -4360.429} C_VEL
LIN {X 0,Y 530.963,Z 372.841,A -85,B 0,C 180,E1 -4363.495,E2 -4363.495} C_VEL
LIN {X 0,Y 530.962,Z 372.846,A -85,B 0,C 180,E1 -4366.507,E2 -4366.507} C_VEL
LIN {X 0,Y 530.986,Z 372.84,A -85,B 0,C 180,E1 -4368.977,E2 -4368.977} C_VEL
LIN {X 0,Y 530.957,Z 372.842,A -85,B 0,C 180,E1 -4371.53,E2 -4371.53} C_VEL
LIN {X 0,Y 530.982,Z 372.845,A -85,B 0,C 180,E1 -4374.383,E2 -4374.383} C_VEL
LIN {X 0,Y 530.974,Z 372.842,A -85,B 0,C 180,E1 -4377.135,E2 -4377.135} C_VEL
LIN {X 0,Y 530.969,Z 372.843,A -85,B 0,C 180,E1 -4379.804,E2 -4379.804} C_VEL
LIN {X 0,Y 531.017,Z 372.844,A -85,B 0,C 180,E1 -4382.467,E2 -4382.467} C_VEL
LIN {X 0,Y 531.009,Z 372.841,A -85,B 0,C 180,E1 -4384.943,E2 -4384.943} C_VEL
LIN {X 0,Y 531.041,Z 372.933,A -85,B 0,C 180,E1 -4386.711,E2 -4386.711} C_VEL
LIN {X 0,Y 532.148,Z 379.87,A -85,B 0,C 180,E1 -4387.972,E2 -4387.972} C_VEL
LIN {X 0,Y 531.854,Z 393.911,A -85,B 0,C 180,E1 -4390.309,E2 -4390.309} C_VEL
LIN {X 0,Y 531.486,Z 410.886,A -85,B 0,C 180,E1 -4393.088,E2 -4393.088} C_VEL
LIN {X 0,Y 531.312,Z 422.795,A -85,B 0,C 180,E1 -4395.005,E2 -4395.005} C_VEL
LIN {X 0,Y 531.586,Z 424.839,A -85,B 0,C 180,E1 -4395.087,E2 -4395.087} C_VEL
LIN {X 0,Y 532.823,Z 433.122,A -85,B 0,C 180,E1 -4395.235,E2 -4395.235} C_VEL
LIN {X 0,Y 532.429,Z 530.728,A -85,B 0,C 180,E1 -4396.572,E2 -4396.572} C_VEL
LIN {X 0,Y 532.245,Z 544.021,A -85,B 0,C 180,E1 -4396.907,E2 -4396.907} C_VEL
LIN {X 0,Y 531.988,Z 557.314,A -85,B 0,C 180,E1 -4397.41,E2 -4397.41} C_VEL
LIN {X 0,Y 531.799,Z 568.826,A -85,B 0,C 180,E1 -4398.009,E2 -4398.009} C_VEL
LIN {X 0,Y 531.509,Z 580.059,A -85,B 0,C 180,E1 -4398.754,E2 -4398.754} C_VEL
LIN {X 0,Y 531.242,Z 590.493,A -85,B 0,C 180,E1 -4399.616,E2 -4399.616} C_VEL
LIN {X 0,Y 531.06,Z 599.021,A -85,B 0,C 180,E1 -4400.479,E2 -4400.479} C_VEL
LIN {X 0,Y 530.886,Z 606.888,A -85,B 0,C 180,E1 -4401.435,E2 -4401.435} C_VEL
LIN {X 0,Y 530.682,Z 614.568,A -85,B 0,C 180,E1 -4402.581,E2 -4402.581} C_VEL
LIN {X 0,Y 530.604,Z 621.647,A -85,B 0,C 180,E1 -4403.918,E2 -4403.918} C_VEL
LIN {X 0,Y 530.459,Z 626.353,A -85,B 0,C 180,E1 -4405.06,E2 -4405.06} C_VEL
LIN {X 0,Y 530.516,Z 629.95,A -85,B 0,C 180,E1 -4406.202,E2 -4406.202} C_VEL
LIN {X 0,Y 530.457,Z 631.804,A -85,B 0,C 180,E1 -4406.962,E2 -4406.962} C_VEL
LIN {X 0,Y 530.41,Z 633.192,A -85,B 0,C 180,E1 -4407.722,E2 -4407.722} C_VEL
LIN {X 0,Y 530.344,Z 634.785,A -85,B 0,C 180,E1 -4409.241,E2 -4409.241} C_VEL
LIN {X 0,Y 530.342,Z 635,A -85,B 0,C 180,E1 -4410,E2 -4410} C_VEL
LIN {X 0,Y 530.361,Z 634.183,A -85,B 0,C 180,E1 -4411.519,E2 -4411.519} C_VEL
LIN {X 0,Y 530.41,Z 633.195,A -85,B 0,C 180,E1 -4412.278,E2 -4412.278} C_VEL
LIN {X 0,Y 530.457,Z 631.807,A -85,B 0,C 180,E1 -4413.038,E2 -4413.038} C_VEL
LIN {X 0,Y 530.522,Z 628.884,A -85,B 0,C 180,E1 -4414.178,E2 -4414.178} C_VEL
LIN {X 0,Y 530.525,Z 624.924,A -85,B 0,C 180,E1 -4415.321,E2 -4415.321} C_VEL
LIN {X 0,Y 530.596,Z 619.238,A -85,B 0,C 180,E1 -4416.579,E2 -4416.579} C_VEL
LIN {X 0,Y 530.758,Z 612.175,A -85,B 0,C 180,E1 -4417.801,E2 -4417.801} C_VEL
LIN {X 0,Y 530.93,Z 603.911,A -85,B 0,C 180,E1 -4418.948,E2 -4418.948} C_VEL
LIN {X 0,Y 531.134,Z 595.439,A -85,B 0,C 180,E1 -4419.905,E2 -4419.905} C_VEL
LIN {X 0,Y 531.393,Z 584.967,A -85,B 0,C 180,E1 -4420.863,E2 -4420.863} C_VEL
LIN {X 0,Y 531.681,Z 573.991,A -85,B 0,C 180,E1 -4421.671,E2 -4421.671} C_VEL
LIN {X 0,Y 531.924,Z 563.24,A -85,B 0,C 180,E1 -4422.301,E2 -4422.301} C_VEL
LIN {X 0,Y 532.13,Z 551.577,A -85,B 0,C 180,E1 -4422.829,E2 -4422.829} C_VEL
LIN {X 0,Y 532.319,Z 538.133,A -85,B 0,C 180,E1 -4423.261,E2 -4423.261} C_VEL
LIN {X 0,Y 532.491,Z 524.833,A -85,B 0,C 180,E1 -4423.524,E2 -4423.524} C_VEL
LIN {X 0,Y 532.701,Z 431.719,A -85,B 0,C 180,E1 -4424.787,E2 -4424.787} C_VEL
LIN {X 0,Y 531.325,Z 423.082,A -85,B 0,C 180,E1 -4424.971,E2 -4424.971} C_VEL
LIN {X 0,Y 531.645,Z 405.068,A -85,B 0,C 180,E1 -4427.862,E2 -4427.862} C_VEL
LIN {X 0,Y 532.086,Z 386.672,A -85,B 0,C 180,E1 -4430.893,E2 -4430.893} C_VEL
LIN {X 0,Y 532.182,Z 379.898,A -85,B 0,C 180,E1 -4432.026,E2 -4432.026} C_VEL
LIN {X 0,Y 531.043,Z 372.955,A -85,B 0,C 180,E1 -4433.289,E2 -4433.289} C_VEL
LIN {X 0,Y 531.015,Z 372.84,A -85,B 0,C 180,E1 -4435.897,E2 -4435.897} C_VEL
LIN {X 0,Y 531,Z 372.838,A -85,B 0,C 180,E1 -4438.455,E2 -4438.455} C_VEL
LIN {X 0,Y 530.965,Z 372.845,A -85,B 0,C 180,E1 -4441.078,E2 -4441.078} C_VEL
LIN {X 0,Y 530.991,Z 372.841,A -85,B 0,C 180,E1 -4443.772,E2 -4443.772} C_VEL
LIN {X 0,Y 530.969,Z 372.841,A -85,B 0,C 180,E1 -4446.557,E2 -4446.557} C_VEL
LIN {X 0,Y 530.983,Z 372.841,A -85,B 0,C 180,E1 -4449.854,E2 -4449.854} C_VEL
LIN {X 0,Y 530.982,Z 372.84,A -85,B 0,C 180,E1 -4452.456,E2 -4452.456} C_VEL
LIN {X 0,Y 530.986,Z 372.842,A -85,B 0,C 180,E1 -4455.62,E2 -4455.62} C_VEL
LIN {X 0,Y 531.017,Z 372.837,A -85,B 0,C 180,E1 -4458.566,E2 -4458.566} C_VEL
LIN {X 0,Y 530.957,Z 372.846,A -85,B 0,C 180,E1 -4461.529,E2 -4461.529} C_VEL
LIN {X 0,Y 530.979,Z 372.841,A -85,B 0,C 180,E1 -4464.382,E2 -4464.382} C_VEL
LIN {X 0,Y 530.969,Z 372.848,A -85,B 0,C 180,E1 -4467.133,E2 -4467.133} C_VEL
LIN {X 0,Y 530.965,Z 372.842,A -85,B 0,C 180,E1 -4469.803,E2 -4469.803} C_VEL
LIN {X 0,Y 531.013,Z 372.839,A -85,B 0,C 180,E1 -4472.466,E2 -4472.466} C_VEL
LIN {X 0,Y 531.003,Z 372.845,A -85,B 0,C 180,E1 -4474.942,E2 -4474.942} C_VEL
LIN {X 0,Y 530.966,Z 372.844,A -85,B 0,C 180,E1 -4478.246,E2 -4478.246} C_VEL
LIN {X 0,Y 530.992,Z 372.844,A -85,B 0,C 180,E1 -4480.677,E2 -4480.677} C_VEL
LIN {X 0,Y 530.987,Z 372.843,A -85,B 0,C 180,E1 -4483.071,E2 -4483.071} C_VEL
LIN {X 0,Y 531.013,Z 372.837,A -85,B 0,C 180,E1 -4485.436,E2 -4485.436} C_VEL
LIN {X 0,Y 531.03,Z 372.84,A -85,B 0,C 180,E1 -4488.549,E2 -4488.549} C_VEL
LIN {X 0,Y 531.051,Z 372.832,A -85,B 0,C 180,E1 -4491.629,E2 -4491.629} C_VEL
LIN {X 0,Y 531.116,Z 372.83,A -85,B 0,C 180,E1 -4494.685,E2 -4494.685} C_VEL
LIN {X 0,Y 531.133,Z 372.822,A -85,B 0,C 180,E1 -4497.725,E2 -4497.725} C_VEL
LIN {X 0,Y 531.148,Z 372.823,A -85,B 0,C 180,E1 -4500.758,E2 -4500.758} C_VEL
LIN {X 0,Y 531.103,Z 372.826,A -85,B 0,C 180,E1 -4503.034,E2 -4503.034} C_VEL
LIN {X 0,Y 531.078,Z 372.834,A -85,B 0,C 180,E1 -4506.077,E2 -4506.077} C_VEL
LIN {X 0,Y 531.025,Z 372.835,A -85,B 0,C 180,E1 -4509.138,E2 -4509.138} C_VEL
LIN {X 0,Y 531.034,Z 372.839,A -85,B 0,C 180,E1 -4512.225,E2 -4512.225} C_VEL
LIN {X 0,Y 530.991,Z 372.84,A -85,B 0,C 180,E1 -4515.35,E2 -4515.35} C_VEL
LIN {X 0,Y 531.01,Z 372.841,A -85,B 0,C 180,E1 -4517.723,E2 -4517.723} C_VEL
LIN {X 0,Y 530.996,Z 372.839,A -85,B 0,C 180,E1 -4520.938,E2 -4520.938} C_VEL
LIN {X 0,Y 530.974,Z 372.846,A -85,B 0,C 180,E1 -4524.225,E2 -4524.225} C_VEL
LIN {X 0,Y 531.007,Z 372.837,A -85,B 0,C 180,E1 -4526.744,E2 -4526.744} C_VEL
LIN {X 0,Y 530.995,Z 372.841,A -85,B 0,C 180,E1 -4529.322,E2 -4529.322} C_VEL
LIN {X 0,Y 530.976,Z 372.846,A -85,B 0,C 180,E1 -4532.104,E2 -4532.104} C_VEL
LIN {X 0,Y 530.986,Z 372.84,A -85,B 0,C 180,E1 -4534.855,E2 -4534.855} C_VEL
LIN {X 0,Y 530.963,Z 372.849,A -85,B 0,C 180,E1 -4537.508,E2 -4537.508} C_VEL
LIN {X 0,Y 530.982,Z 372.84,A -85,B 0,C 180,E1 -4540.433,E2 -4540.433} C_VEL
LIN {X 0,Y 530.968,Z 372.846,A -85,B 0,C 180,E1 -4543.283,E2 -4543.283} C_VEL
LIN {X 0,Y 530.961,Z 372.849,A -85,B 0,C 180,E1 -4543.575,E2 -4543.575} C_VEL
LIN {X 0,Y 530.287,Z 372.929,A -85,B 0,C 180,E1 -4544.209,E2 -4544.209} C_VEL
LIN {X 0,Y 527.438,Z 373.286,A -85,B 0,C 180,E1 -4545.238,E2 -4545.238} C_VEL
LIN {X 0,Y 525.034,Z 373.583,A -85,B 0,C 180,E1 -4546.066,E2 -4546.066} C_VEL
LIN {X 0,Y 524.001,Z 373.71,A -85,B 0,C 180,E1 -4546.706,E2 -4546.706} C_VEL
LIN {X 0,Y 523.917,Z 373.721,A -85,B 0,C 180,E1 -4546.922,E2 -4546.922} C_VEL
LIN {X 0,Y 523.977,Z 373.715,A -85,B 0,C 180,E1 -4549.924,E2 -4549.924} C_VEL
LIN {X 0,Y 523.911,Z 373.722,A -85,B 0,C 180,E1 -4552.869,E2 -4552.869} C_VEL
LIN {X 0,Y 523.944,Z 373.72,A -85,B 0,C 180,E1 -4555.711,E2 -4555.711} C_VEL
LIN {X 0,Y 523.923,Z 373.719,A -85,B 0,C 180,E1 -4558.457,E2 -4558.457} C_VEL
LIN {X 0,Y 523.939,Z 373.724,A -85,B 0,C 180,E1 -4561.126,E2 -4561.126} C_VEL
LIN {X 0,Y 523.985,Z 373.711,A -85,B 0,C 180,E1 -4563.981,E2 -4563.981} C_VEL
LIN {X 0,Y 523.927,Z 373.718,A -85,B 0,C 180,E1 -4566.271,E2 -4566.271} C_VEL
LIN {X 0,Y 523.946,Z 373.719,A -85,B 0,C 180,E1 -4568.767,E2 -4568.767} C_VEL
LIN {X 0,Y 523.951,Z 373.721,A -85,B 0,C 180,E1 -4571.221,E2 -4571.221} C_VEL
LIN {X 0,Y 523.938,Z 373.718,A -85,B 0,C 180,E1 -4573.639,E2 -4573.639} C_VEL
LIN {X 0,Y 523.941,Z 373.717,A -85,B 0,C 180,E1 -4576.028,E2 -4576.028} C_VEL
LIN {X 0,Y 524.015,Z 373.711,A -85,B 0,C 180,E1 -4578.394,E2 -4578.394} C_VEL
LIN {X 0,Y 524.05,Z 373.904,A -85,B 0,C 180,E1 -4581.371,E2 -4581.371} C_VEL
LIN {X 0,Y 524.895,Z 379.901,A -85,B 0,C 180,E1 -4582.545,E2 -4582.545} C_VEL
LIN {X 0,Y 524.658,Z 390.08,A -85,B 0,C 180,E1 -4584.427,E2 -4584.427} C_VEL
LIN {X 0,Y 524.284,Z 406.986,A -85,B 0,C 180,E1 -4587.503,E2 -4587.503} C_VEL
LIN {X 0,Y 524.34,Z 409.453,A -85,B 0,C 180,E1 -4587.887,E2 -4587.887} C_VEL
LIN {X 0,Y 525.928,Z 418.859,A -85,B 0,C 180,E1 -4588.085,E2 -4588.085} C_VEL
LIN {X 0,Y 525.491,Z 516.743,A -85,B 0,C 180,E1 -4589.449,E2 -4589.449} C_VEL
LIN {X 0,Y 525.318,Z 530.411,A -85,B 0,C 180,E1 -4589.808,E2 -4589.808} C_VEL
LIN {X 0,Y 525.088,Z 542.715,A -85,B 0,C 180,E1 -4590.287,E2 -4590.287} C_VEL
LIN {X 0,Y 524.799,Z 553.749,A -85,B 0,C 180,E1 -4590.863,E2 -4590.863} C_VEL
LIN {X 0,Y 524.474,Z 565.221,A -85,B 0,C 180,E1 -4591.632,E2 -4591.632} C_VEL
LIN {X 0,Y 524.206,Z 575.556,A -85,B 0,C 180,E1 -4592.497,E2 -4592.497} C_VEL
LIN {X 0,Y 523.955,Z 584.906,A -85,B 0,C 180,E1 -4593.46,E2 -4593.46} C_VEL
LIN {X 0,Y 523.746,Z 593.932,A -85,B 0,C 180,E1 -4594.618,E2 -4594.618} C_VEL
LIN {X 0,Y 523.609,Z 601.23,A -85,B 0,C 180,E1 -4595.777,E2 -4595.777} C_VEL
LIN {X 0,Y 523.488,Z 607.106,A -85,B 0,C 180,E1 -4596.94,E2 -4596.94} C_VEL
LIN {X 0,Y 523.441,Z 611.749,A -85,B 0,C 180,E1 -4598.104,E2 -4598.104} C_VEL
LIN {X 0,Y 523.328,Z 615.304,A -85,B 0,C 180,E1 -4599.273,E2 -4599.273} C_VEL
LIN {X 0,Y 523.32,Z 617.103,A -85,B 0,C 180,E1 -4600.054,E2 -4600.054} C_VEL
LIN {X 0,Y 523.362,Z 619.183,A -85,B 0,C 180,E1 -4601.396,E2 -4601.396} C_VEL
LIN {X 0,Y 523.281,Z 619.978,A -85,B 0,C 180,E1 -4602.409,E2 -4602.409} C_VEL
LIN {X 0,Y 523.268,Z 620.088,A -85,B 0,C 180,E1 -4603.198,E2 -4603.198} C_VEL
LIN {X 0,Y 523.294,Z 619.79,A -85,B 0,C 180,E1 -4603.989,E2 -4603.989} C_VEL
LIN {X 0,Y 523.3,Z 619.091,A -85,B 0,C 180,E1 -4604.783,E2 -4604.783} C_VEL
LIN {X 0,Y 523.251,Z 617.955,A -85,B 0,C 180,E1 -4605.582,E2 -4605.582} C_VEL
LIN {X 0,Y 523.327,Z 615.399,A -85,B 0,C 180,E1 -4606.782,E2 -4606.782} C_VEL
LIN {X 0,Y 523.421,Z 611.747,A -85,B 0,C 180,E1 -4607.988,E2 -4607.988} C_VEL
LIN {X 0,Y 523.512,Z 606.87,A -85,B 0,C 180,E1 -4609.202,E2 -4609.202} C_VEL
LIN {X 0,Y 523.615,Z 600.596,A -85,B 0,C 180,E1 -4610.424,E2 -4610.424} C_VEL
LIN {X 0,Y 523.818,Z 592.686,A -85,B 0,C 180,E1 -4611.651,E2 -4611.651} C_VEL
LIN {X 0,Y 524.046,Z 584.248,A -85,B 0,C 180,E1 -4612.702,E2 -4612.702} C_VEL
LIN {X 0,Y 524.274,Z 574.244,A -85,B 0,C 180,E1 -4613.712,E2 -4613.712} C_VEL
LIN {X 0,Y 524.534,Z 564.124,A -85,B 0,C 180,E1 -4614.541,E2 -4614.541} C_VEL
LIN {X 0,Y 524.833,Z 553.093,A -85,B 0,C 180,E1 -4615.266,E2 -4615.266} C_VEL
LIN {X 0,Y 525.11,Z 540.733,A -85,B 0,C 180,E1 -4615.889,E2 -4615.889} C_VEL
LIN {X 0,Y 525.4,Z 527.679,A -85,B 0,C 180,E1 -4616.369,E2 -4616.369} C_VEL
LIN {X 0,Y 525.539,Z 514.739,A -85,B 0,C 180,E1 -4616.678,E2 -4616.678} C_VEL
LIN {X 0,Y 525.909,Z 418.948,A -85,B 0,C 180,E1 -4618.005,E2 -4618.005} C_VEL
LIN {X 0,Y 524.281,Z 409.48,A -85,B 0,C 180,E1 -4618.203,E2 -4618.203} C_VEL
LIN {X 0,Y 524.286,Z 406.752,A -85,B 0,C 180,E1 -4618.634,E2 -4618.634} C_VEL
LIN {X 0,Y 524.681,Z 389.822,A -85,B 0,C 180,E1 -4621.717,E2 -4621.717} C_VEL
LIN {X 0,Y 524.927,Z 379.739,A -85,B 0,C 180,E1 -4623.577,E2 -4623.577} C_VEL
LIN {X 0,Y 523.967,Z 373.794,A -85,B 0,C 180,E1 -4624.774,E2 -4624.774} C_VEL
LIN {X 0,Y 523.912,Z 373.724,A -85,B 0,C 180,E1 -4627.678,E2 -4627.678} C_VEL
LIN {X 0,Y 523.964,Z 373.715,A -85,B 0,C 180,E1 -4630.133,E2 -4630.133} C_VEL
LIN {X 0,Y 523.921,Z 373.725,A -85,B 0,C 180,E1 -4633.166,E2 -4633.166} C_VEL
LIN {X 0,Y 523.937,Z 373.718,A -85,B 0,C 180,E1 -4635.772,E2 -4635.772} C_VEL
LIN {X 0,Y 523.964,Z 373.717,A -85,B 0,C 180,E1 -4638.91,E2 -4638.91} C_VEL
LIN {X 0,Y 523.913,Z 373.719,A -85,B 0,C 180,E1 -4641.898,E2 -4641.898} C_VEL
LIN {X 0,Y 523.933,Z 373.722,A -85,B 0,C 180,E1 -4644.908,E2 -4644.908} C_VEL
LIN {X 0,Y 523.936,Z 373.718,A -85,B 0,C 180,E1 -4647.677,E2 -4647.677} C_VEL
LIN {X 0,Y 523.962,Z 373.712,A -85,B 0,C 180,E1 -4650.673,E2 -4650.673} C_VEL
LIN {X 0,Y 523.97,Z 373.713,A -85,B 0,C 180,E1 -4653.728,E2 -4653.728} C_VEL
LIN {X 0,Y 523.942,Z 373.717,A -85,B 0,C 180,E1 -4656.271,E2 -4656.271} C_VEL
LIN {X 0,Y 523.945,Z 373.719,A -85,B 0,C 180,E1 -4658.767,E2 -4658.767} C_VEL
LIN {X 0,Y 523.948,Z 373.718,A -85,B 0,C 180,E1 -4661.221,E2 -4661.221} C_VEL
LIN {X 0,Y 523.933,Z 373.718,A -85,B 0,C 180,E1 -4663.639,E2 -4663.639} C_VEL
LIN {X 0,Y 523.932,Z 373.715,A -85,B 0,C 180,E1 -4666.028,E2 -4666.028} C_VEL
LIN {X 0,Y 524.002,Z 373.711,A -85,B 0,C 180,E1 -4668.394,E2 -4668.394} C_VEL
LIN {X 0,Y 524,Z 373.71,A -85,B 0,C 180,E1 -4671.516,E2 -4671.516} C_VEL
LIN {X 0,Y 524.091,Z 373.7,A -85,B 0,C 180,E1 -4674.614,E2 -4674.614} C_VEL
LIN {X 0,Y 524.104,Z 373.695,A -85,B 0,C 180,E1 -4677.695,E2 -4677.695} C_VEL
LIN {X 0,Y 524.119,Z 373.701,A -85,B 0,C 180,E1 -4680.768,E2 -4680.768} C_VEL
LIN {X 0,Y 524.069,Z 373.702,A -85,B 0,C 180,E1 -4683.075,E2 -4683.075} C_VEL
LIN {X 0,Y 524.038,Z 373.705,A -85,B 0,C 180,E1 -4686.159,E2 -4686.159} C_VEL
LIN {X 0,Y 523.996,Z 373.71,A -85,B 0,C 180,E1 -4689.262,E2 -4689.262} C_VEL
LIN {X 0,Y 524.015,Z 373.706,A -85,B 0,C 180,E1 -4691.752,E2 -4691.752} C_VEL
LIN {X 0,Y 523.983,Z 373.715,A -85,B 0,C 180,E1 -4695.053,E2 -4695.053} C_VEL
LIN {X 0,Y 523.956,Z 373.713,A -85,B 0,C 180,E1 -4697.969,E2 -4697.969} C_VEL
LIN {X 0,Y 523.965,Z 373.717,A -85,B 0,C 180,E1 -4700.41,E2 -4700.41} C_VEL
LIN {X 0,Y 523.936,Z 373.721,A -85,B 0,C 180,E1 -4702.893,E2 -4702.893} C_VEL
LIN {X 0,Y 523.978,Z 373.712,A -85,B 0,C 180,E1 -4706.021,E2 -4706.021} C_VEL
LIN {X 0,Y 523.934,Z 373.722,A -85,B 0,C 180,E1 -4708.875,E2 -4708.875} C_VEL
LIN {X 0,Y 523.924,Z 373.717,A -85,B 0,C 180,E1 -4711.544,E2 -4711.544} C_VEL
LIN {X 0,Y 523.94,Z 373.72,A -85,B 0,C 180,E1 -4714.29,E2 -4714.29} C_VEL
LIN {X 0,Y 523.907,Z 373.721,A -85,B 0,C 180,E1 -4717.132,E2 -4717.132} C_VEL
LIN {X 0,Y 523.963,Z 373.716,A -85,B 0,C 180,E1 -4720.135,E2 -4720.135} C_VEL
LIN {X 0,Y 523.922,Z 373.72,A -85,B 0,C 180,E1 -4723.167,E2 -4723.167} C_VEL
LIN {X 0,Y 523.937,Z 373.715,A -85,B 0,C 180,E1 -4725.773,E2 -4725.773} C_VEL
LIN {X 0,Y 523.941,Z 373.718,A -85,B 0,C 180,E1 -4728.909,E2 -4728.909} C_VEL
LIN {X 0,Y 523.915,Z 373.721,A -85,B 0,C 180,E1 -4731.899,E2 -4731.899} C_VEL
LIN {X 0,Y 523.939,Z 373.72,A -85,B 0,C 180,E1 -4734.909,E2 -4734.909} C_VEL
LIN {X 0,Y 523.942,Z 373.717,A -85,B 0,C 180,E1 -4737.679,E2 -4737.679} C_VEL
LIN {X 0,Y 523.954,Z 373.722,A -85,B 0,C 180,E1 -4740.677,E2 -4740.677} C_VEL
LIN {X 0,Y 523.978,Z 373.715,A -85,B 0,C 180,E1 -4743.73,E2 -4743.73} C_VEL
LIN {X 0,Y 523.968,Z 373.804,A -85,B 0,C 180,E1 -4746.535,E2 -4746.535} C_VEL
LIN {X 0,Y 525.132,Z 380.276,A -85,B 0,C 180,E1 -4747.745,E2 -4747.745} C_VEL
LIN {X 0,Y 524.991,Z 391.036,A -85,B 0,C 180,E1 -4749.568,E2 -4749.568} C_VEL
LIN {X 0,Y 524.612,Z 408.363,A -85,B 0,C 180,E1 -4752.457,E2 -4752.457} C_VEL
LIN {X 0,Y 524.303,Z 422.974,A -85,B 0,C 180,E1 -4754.824,E2 -4754.824} C_VEL
LIN {X 0,Y 525.955,Z 433.6,A -85,B 0,C 180,E1 -4755.046,E2 -4755.046} C_VEL
LIN {X 0,Y 525.533,Z 530.588,A -85,B 0,C 180,E1 -4756.392,E2 -4756.392} C_VEL
LIN {X 0,Y 525.325,Z 543.893,A -85,B 0,C 180,E1 -4756.731,E2 -4756.731} C_VEL
LIN {X 0,Y 525.042,Z 557.193,A -85,B 0,C 180,E1 -4757.241,E2 -4757.241} C_VEL
LIN {X 0,Y 524.809,Z 569.714,A -85,B 0,C 180,E1 -4757.909,E2 -4757.909} C_VEL
LIN {X 0,Y 524.508,Z 581.239,A -85,B 0,C 180,E1 -4758.699,E2 -4758.699} C_VEL
LIN {X 0,Y 524.224,Z 591.426,A -85,B 0,C 180,E1 -4759.573,E2 -4759.573} C_VEL
LIN {X 0,Y 523.966,Z 600.589,A -85,B 0,C 180,E1 -4760.543,E2 -4760.543} C_VEL
LIN {X 0,Y 523.747,Z 609.515,A -85,B 0,C 180,E1 -4761.706,E2 -4761.706} C_VEL
LIN {X 0,Y 523.583,Z 616.696,A -85,B 0,C 180,E1 -4762.868,E2 -4762.868} C_VEL
LIN {X 0,Y 523.523,Z 623.235,A -85,B 0,C 180,E1 -4764.222,E2 -4764.222} C_VEL
LIN {X 0,Y 523.36,Z 627.558,A -85,B 0,C 180,E1 -4765.379,E2 -4765.379} C_VEL
LIN {X 0,Y 523.443,Z 629.848,A -85,B 0,C 180,E1 -4766.151,E2 -4766.151} C_VEL
LIN {X 0,Y 523.367,Z 631.703,A -85,B 0,C 180,E1 -4766.921,E2 -4766.921} C_VEL
LIN {X 0,Y 523.334,Z 633.093,A -85,B 0,C 180,E1 -4767.691,E2 -4767.691} C_VEL
LIN {X 0,Y 523.25,Z 634.69,A -85,B 0,C 180,E1 -4769.231,E2 -4769.231} C_VEL
LIN {X 0,Y 523.246,Z 634.906,A -85,B 0,C 180,E1 -4770,E2 -4770} C_VEL
LIN {X 0,Y 523.274,Z 634.087,A -85,B 0,C 180,E1 -4771.539,E2 -4771.539} C_VEL
LIN {X 0,Y 523.334,Z 633.096,A -85,B 0,C 180,E1 -4772.309,E2 -4772.309} C_VEL
